Yaskawa INFORM job: CONTOUR2.JBI

/JOB
//NAME CONTOUR2
//POS
///NPOS 9848,0,0,0,0,0
///TOOL 0
///POSTYPE PULSE
///PULSE
C00000=-41004,59868,4099,4900,-34257,16705
C00001=-41004,59868,1099,4900,-34257,16705
C00002=-41004,64596,1380,5213,-31659,16463
C00003=-41004,59868,1099,4900,-34257,16705
C00004=-41004,59868,9099,4900,-34257,16705
C00005=3811,31631,-25134,676,-27450,-2228
C00006=3865,31716,-25032,668,-27483,-2249
C00007=3865,31716,-29032,668,-27483,-2249
C00008=3835,31810,-28918,671,-27518,-2237
C00009=3597,31820,-28908,705,-27519,-2144
C00010=3355,31766,-28975,741,-27496,-2051
C00011=3123,31694,-29064,775,-27467,-1961
C00012=2902,31602,-29176,808,-27431,-1876
C00013=2696,31482,-29322,839,-27385,-1796
C00014=2515,31319,-29520,866,-27323,-1727
C00015=2374,31161,-29713,888,-27263,-1673
C00016=2389,31321,-29519,885,-27322,-1678
C00017=2255,31496,-29308,902,-27386,-1624
C00018=2187,31630,-29147,910,-27435,-1597
C00019=2310,31450,-29364,894,-27369,-1646
C00020=2453,31290,-29556,876,-27311,-1703
C00021=2629,31465,-29344,848,-27378,-1770
C00022=2553,31625,-29151,858,-27436,-1740
C00023=2441,31812,-28926,872,-27504,-1694
C00024=2353,32012,-28684,882,-27578,-1659
C00025=2314,32240,-28409,885,-27661,-1642
C00026=2304,32475,-28124,884,-27749,-1636
C00027=2314,32706,-27845,880,-27834,-1639
C00028=2326,32679,-27878,879,-27824,-1644
C00029=2316,32448,-28157,883,-27739,-1641
C00030=2336,32210,-28445,883,-27651,-1651
C00031=2378,31984,-28718,879,-27567,-1669
C00032=2473,31787,-28955,867,-27496,-1707
C00033=2590,31603,-29177,853,-27428,-1754
C00034=2757,31554,-29235,829,-27412,-1819
C00035=2747,31685,-29077,829,-27460,-1815
C00036=2622,31865,-28860,845,-27526,-1765
C00037=2549,32074,-28608,854,-27603,-1735
C00038=2549,31957,-28749,855,-27559,-1736
C00039=2637,31757,-28991,844,-27486,-1771
C00040=2729,31601,-29178,833,-27429,-1808
C00041=2605,31782,-28960,849,-27495,-1759
C00042=2520,31985,-28716,859,-27569,-1724
C00043=2477,32210,-28444,863,-27652,-1706
C00044=2487,32441,-28165,859,-27738,-1708
C00045=2486,32674,-27883,856,-27824,-1706
C00046=2496,32905,-27604,853,-27910,-1708
C00047=2495,33138,-27322,850,-27996,-1706
C00048=2455,33357,-27057,854,-28077,-1689
C00049=2239,33295,-27134,885,-28051,-1605
C00050=2171,33103,-27367,896,-27979,-1580
C00051=2146,32876,-27642,902,-27895,-1572
C00052=2089,32656,-27907,913,-27813,-1551
C00053=2047,32433,-28178,921,-27730,-1537
C00054=2015,32207,-28451,928,-27646,-1526
C00055=2004,31976,-28730,933,-27561,-1523
C00056=2032,31743,-29011,931,-27475,-1536
C00057=2100,31532,-29266,924,-27397,-1564
C00058=2192,31334,-29505,913,-27325,-1601
C00059=2314,31152,-29724,897,-27259,-1650
C00060=2441,30973,-29940,881,-27194,-1701
C00061=2538,31160,-29713,865,-27264,-1737
C00062=2713,31335,-29500,838,-27330,-1804
C00063=2925,31445,-29366,806,-27373,-1885
C00064=3143,31543,-29246,774,-27412,-1970
C00065=3375,31616,-29157,739,-27441,-2059
C00066=3618,31670,-29089,704,-27463,-2153
C00067=3865,31716,-29032,668,-27483,-2249
C00068=3865,31716,-27632,668,-27483,-2249
C00069=3997,31675,-25080,649,-27469,-2301
C00070=3997,31675,-29080,649,-27469,-2301
C00071=3629,31643,-29122,703,-27453,-2158
C00072=3265,31552,-29234,756,-27416,-2017
C00073=3117,31368,-29458,779,-27346,-1961
C00074=2827,31365,-29463,821,-27343,-1848
C00075=2560,31123,-29757,862,-27250,-1746
C00076=2498,30791,-30159,875,-27127,-1724
C00077=2587,30462,-30556,865,-27006,-1761
C00078=2678,30133,-30954,855,-26885,-1799
C00079=2799,29820,-31331,841,-26770,-1848
C00080=2795,29751,-31415,842,-26744,-1847
C00081=2700,29995,-31120,854,-26834,-1808
C00082=2657,29651,-31536,864,-26706,-1794
C00083=2597,29318,-31939,876,-26583,-1774
C00084=2683,28990,-32335,867,-26462,-1809
C00085=2723,28642,-32756,865,-26333,-1827
C00086=2815,28557,-32857,852,-26303,-1863
C00087=2847,28244,-33236,851,-26187,-1878
C00088=2952,27925,-33622,839,-26069,-1921
C00089=3213,27690,-33905,802,-25984,-2023
C00090=3033,27904,-33647,827,-26062,-1952
C00091=2962,28220,-33265,834,-26179,-1922
C00092=2963,28089,-33423,835,-26130,-1924
C00093=3143,27897,-33654,810,-26061,-1995
C00094=3098,28244,-33236,814,-26189,-1975
C00095=3076,28338,-33122,816,-26223,-1966
C00096=3042,28684,-32704,817,-26351,-1950
C00097=3058,29035,-32280,811,-26481,-1954
C00098=3108,29326,-31927,801,-26589,-1971
C00099=3276,29624,-31566,773,-26701,-2034
C00100=3295,29634,-31554,770,-26705,-2041
C00101=3459,29782,-31375,745,-26761,-2103
C00102=3564,30094,-30996,726,-26878,-2142
C00103=3359,30318,-30727,754,-26959,-2061
C00104=3037,30467,-30548,800,-27011,-1935
C00105=3111,30271,-30785,791,-26939,-1965
C00106=3111,29941,-31184,794,-26817,-1968
C00107=3089,29614,-31579,801,-26696,-1962
C00108=3061,29461,-31764,806,-26639,-1952
C00109=3123,29801,-31353,794,-26765,-1974
C00110=3092,30139,-30945,795,-26890,-1959
C00111=2965,30424,-30600,810,-26995,-1908
C00112=2876,30690,-30279,821,-27093,-1872
C00113=2659,30936,-29983,850,-27182,-1786
C00114=2871,30740,-30218,821,-27111,-1869
C00115=3081,30482,-30530,793,-27018,-1953
C00116=3405,30337,-30703,747,-26967,-2079
C00117=3629,30413,-30610,714,-26997,-2165
C00118=3603,30113,-30974,720,-26885,-2157
C00119=3702,29893,-31239,708,-26804,-2197
C00120=4073,29908,-31220,653,-26812,-2340
C00121=4409,29785,-31366,605,-26769,-2471
C00122=4667,29549,-31651,569,-26683,-2572
C00123=4682,29665,-31511,566,-26727,-2577
C00124=4727,30001,-31105,556,-26852,-2593
C00125=4672,30326,-30711,562,-26973,-2570
C00126=4650,30631,-30342,563,-27086,-2559
C00127=4609,30958,-29945,566,-27208,-2542
C00128=4531,31274,-29563,575,-27324,-2510
C00129=4306,31488,-29305,606,-27402,-2422
C00130=3997,31675,-29080,649,-27469,-2301
C00131=3997,31675,-27680,649,-27469,-2301
C00132=4043,31695,-25057,642,-27476,-2318
C00133=4043,31695,-29057,642,-27476,-2318
C00134=5780,31150,-29707,394,-27289,-2995
C00135=5625,31340,-29477,415,-27359,-2934
C00136=3945,31835,-28888,655,-27528,-2280
C00137=5709,31371,-29439,403,-27371,-2966
C00138=6652,32744,-27767,260,-27893,-3328
C00139=6753,34511,-25621,239,-28558,-3363
C00140=6453,36318,-23427,276,-29233,-3243
C00141=6578,35948,-23875,259,-29096,-3292
C00142=6792,34132,-26080,234,-28416,-3379
C00143=6645,32383,-28206,262,-27758,-3326
C00144=7120,32806,-27689,192,-27921,-3510
C00145=6925,34048,-26182,216,-28386,-3431
C00146=6644,35901,-23931,250,-29079,-3318
C00147=5803,37019,-22583,363,-29488,-2986
C00148=3963,36746,-22938,616,-29357,-2262
C00149=2129,36463,-23304,868,-29224,-1540
C00150=289,36189,-23660,1121,-29094,-816
C00151=213,34463,-25744,1154,-28457,-802
C00152=323,33186,-27283,1156,-27988,-857
C00153=1338,31882,-28849,1029,-27519,-1265
C00154=2465,30575,-30421,882,-27047,-1713
C00155=1969,32162,-28506,936,-27629,-1508
C00156=1600,32867,-27657,980,-27886,-1359
C00157=996,33032,-27463,1063,-27939,-1121
C00158=1818,33311,-27119,944,-28052,-1440
C00159=1626,33396,-27018,970,-28081,-1365
C00160=1314,33620,-26749,1011,-28160,-1241
C00161=796,33812,-26524,1082,-28224,-1036
C00162=1636,32812,-27724,976,-27865,-1373
C00163=721,33056,-27436,1102,-27945,-1014
C00164=1464,34245,-25993,983,-28393,-1295
C00165=1936,35230,-24798,907,-28764,-1473
C00166=2213,35790,-24117,863,-28976,-1578
C00167=3722,35571,-24365,657,-28916,-2172
C00168=4244,35600,-24324,585,-28934,-2377
C00169=2395,35403,-24583,842,-28835,-1652
C00170=3210,35322,-24671,730,-28816,-1972
C00171=3567,35347,-24638,680,-28830,-2113
C00172=2031,34952,-25133,897,-28662,-1512
C00173=3721,35166,-23455,660,-28765,-2174
C00174=-41004,59868,4099,4900,-34257,16705
C00175=-41004,59868,1099,4900,-34257,16705
C00176=-41004,64596,1380,5213,-31659,16463
C00177=-41004,59868,1099,4900,-34257,16705
C00178=-41004,59868,9099,4900,-34257,16705
C00179=3721,35166,-20855,660,-28765,-2174
C00180=3721,35166,-24855,660,-28765,-2174
C00181=2130,35067,-24992,882,-28706,-1550
C00182=3955,35232,-24773,627,-28793,-2265
C00183=5703,35515,-24411,383,-28922,-2950
C00184=5623,36481,-23238,390,-29283,-2916
C00185=6165,34818,-25253,321,-28666,-3133
C00186=6218,33011,-27446,321,-27989,-3159
C00187=5066,32366,-28237,490,-27736,-2713
C00188=6014,32285,-28329,354,-27715,-3082
C00189=4649,33272,-27142,543,-28070,-2546
C00190=3598,34047,-26212,686,-28347,-2132
C00191=3164,33192,-27250,755,-28024,-1967
C00192=4473,31982,-28706,578,-27588,-2484
C00193=6195,31948,-28737,329,-27591,-3153
C00194=6280,32014,-28656,317,-27616,-3186
C00195=4570,31861,-28851,565,-27544,-2522
C00196=4080,32067,-28606,634,-27615,-2331
C00197=3506,32938,-27555,709,-27934,-2102
C00198=3001,33034,-27443,780,-27963,-1905
C00199=2855,33000,-27485,801,-27949,-1848
C00200=4043,31695,-29057,642,-27476,-2318
C00201=4043,31695,-27657,642,-27476,-2318
C00202=4163,31799,-24930,624,-27516,-2364
C00203=4163,31799,-28930,624,-27516,-2364
C00204=4084,31834,-28888,635,-27529,-2334
C00205=4008,31876,-28837,646,-27544,-2304
C00206=3930,31915,-28790,657,-27557,-2273
C00207=3853,31954,-28744,668,-27571,-2243
C00208=3786,32011,-28676,677,-27591,-2217
C00209=3763,32036,-28645,680,-27601,-2208
C00210=3832,31988,-28702,670,-27584,-2235
C00211=3909,31948,-28751,659,-27569,-2265
C00212=3987,31909,-28797,649,-27556,-2295
C00213=4064,31869,-28845,638,-27542,-2325
C00214=4142,31831,-28890,627,-27528,-2356
C00215=4222,31800,-28928,616,-27517,-2387
C00216=4302,31768,-28966,604,-27506,-2419
C00217=4382,31737,-29004,593,-27495,-2450
C00218=4465,31712,-29033,581,-27487,-2482
C00219=4547,31688,-29062,569,-27479,-2514
C00220=4630,31664,-29090,558,-27471,-2547
C00221=4713,31639,-29120,546,-27462,-2579
C00222=4798,31621,-29141,534,-27456,-2612
C00223=4883,31604,-29161,522,-27450,-2645
C00224=4968,31586,-29182,509,-27445,-2678
C00225=5053,31569,-29203,497,-27439,-2711
C00226=5140,31557,-29217,485,-27435,-2745
C00227=5225,31540,-29237,472,-27430,-2778
C00228=5314,31534,-29244,459,-27428,-2813
C00229=5403,31528,-29251,447,-27427,-2847
C00230=5495,31531,-29246,433,-27429,-2883
C00231=5589,31545,-29228,419,-27435,-2919
C00232=5684,31559,-29211,406,-27441,-2956
C00233=5773,31582,-29183,392,-27450,-2991
C00234=5862,31604,-29155,379,-27459,-3025
C00235=5946,31635,-29117,367,-27472,-3058
C00236=6027,31672,-29072,355,-27486,-3089
C00237=6103,31716,-29019,344,-27503,-3118
C00238=6174,31767,-28957,333,-27523,-3145
C00239=6196,31760,-28964,330,-27521,-3154
C00240=6126,31707,-29029,341,-27500,-3127
C00241=6052,31660,-29086,352,-27482,-3098
C00242=5973,31620,-29135,363,-27466,-3068
C00243=5890,31589,-29174,376,-27454,-3036
C00244=5800,31566,-29202,389,-27445,-3001
C00245=5711,31544,-29229,402,-27435,-2967
C00246=5616,31530,-29247,416,-27430,-2930
C00247=5522,31516,-29264,429,-27424,-2893
C00248=5427,31502,-29281,443,-27418,-2857
C00249=5338,31509,-29274,456,-27419,-2822
C00250=5249,31515,-29267,469,-27421,-2788
C00251=5162,31526,-29254,482,-27424,-2754
C00252=5077,31544,-29233,494,-27430,-2721
C00253=4992,31561,-29213,506,-27435,-2687
C00254=4907,31578,-29192,518,-27441,-2654
C00255=4822,31596,-29172,530,-27447,-2621
C00256=4736,31613,-29152,543,-27452,-2588
C00257=4652,31631,-29130,555,-27458,-2555
C00258=4569,31655,-29101,567,-27467,-2523
C00259=4486,31680,-29072,578,-27475,-2491
C00260=4404,31704,-29043,590,-27483,-2458
C00261=4323,31734,-29007,602,-27494,-2427
C00262=4241,31761,-28975,613,-27503,-2395
C00263=4163,31799,-28930,624,-27516,-2364
C00264=4163,31799,-27530,624,-27516,-2364
C00265=4231,31880,-24831,614,-27547,-2390
C00266=4231,31880,-28831,614,-27547,-2390
C00267=4158,31906,-28799,624,-27556,-2362
C00268=4087,31940,-28759,634,-27568,-2334
C00269=4017,31974,-28719,644,-27580,-2307
C00270=3946,32007,-28678,654,-27592,-2279
C00271=3878,32048,-28629,663,-27606,-2252
C00272=3808,32082,-28589,673,-27618,-2225
C00273=3738,32118,-28546,683,-27631,-2197
C00274=3669,32157,-28500,692,-27645,-2170
C00275=3604,32205,-28442,701,-27662,-2145
C00276=3536,32245,-28393,711,-27676,-2118
C00277=3474,32295,-28333,719,-27694,-2094
C00278=3419,32349,-28269,726,-27713,-2072
C00279=3360,32401,-28207,734,-27732,-2048
C00280=3308,32456,-28140,741,-27752,-2028
C00281=3261,32514,-28070,747,-27773,-2009
C00282=3215,32573,-27999,753,-27795,-1991
C00283=3179,32637,-27922,758,-27818,-1976
C00284=3142,32701,-27845,763,-27841,-1962
C00285=3098,32760,-27773,768,-27863,-1944
C00286=3061,32824,-27696,773,-27886,-1929
C00287=3041,32881,-27628,775,-27907,-1921
C00288=3081,32819,-27702,770,-27885,-1937
C00289=3124,32759,-27775,765,-27863,-1954
C00290=3163,32696,-27850,760,-27840,-1970
C00291=3200,32632,-27927,755,-27816,-1985
C00292=3245,32573,-27999,749,-27795,-2002
C00293=3289,32514,-28070,743,-27773,-2020
C00294=3341,32458,-28137,737,-27753,-2041
C00295=3393,32403,-28204,730,-27733,-2061
C00296=3451,32351,-28266,722,-27715,-2084
C00297=3510,32299,-28328,714,-27696,-2108
C00298=3576,32251,-28386,705,-27679,-2133
C00299=3643,32209,-28436,695,-27664,-2160
C00300=3709,32162,-28492,686,-27647,-2186
C00301=3777,32122,-28541,677,-27633,-2213
C00302=3847,32088,-28582,667,-27621,-2240
C00303=3916,32047,-28631,658,-27606,-2267
C00304=3986,32013,-28671,648,-27595,-2294
C00305=4054,31973,-28720,638,-27580,-2321
C00306=4125,31939,-28760,628,-27568,-2349
C00307=4198,31912,-28792,618,-27559,-2377
C00308=4269,31880,-28831,608,-27548,-2405
C00309=4342,31852,-28864,598,-27538,-2434
C00310=4415,31824,-28897,588,-27528,-2462
C00311=4486,31792,-28936,578,-27517,-2490
C00312=4559,31765,-28968,567,-27508,-2519
C00313=4633,31739,-29000,557,-27498,-2547
C00314=4707,31714,-29029,546,-27490,-2576
C00315=4782,31693,-29054,535,-27483,-2605
C00316=4856,31668,-29083,525,-27474,-2634
C00317=4895,31655,-29099,519,-27470,-2650
C00318=4818,31667,-29085,531,-27474,-2619
C00319=4743,31690,-29058,541,-27481,-2590
C00320=4668,31713,-29030,552,-27489,-2561
C00321=4594,31736,-29004,562,-27497,-2532
C00322=4521,31763,-28971,573,-27507,-2504
C00323=4448,31791,-28937,583,-27516,-2475
C00324=4375,31820,-28903,593,-27526,-2447
C00325=4302,31846,-28871,604,-27535,-2418
C00326=4231,31880,-28831,614,-27547,-2390
C00327=4231,31880,-27431,614,-27547,-2390
C00328=3770,31874,-24841,680,-27541,-2211
C00329=3770,31874,-28841,680,-27541,-2211
C00330=3645,31974,-28721,697,-27577,-2162
C00331=3526,32078,-28596,713,-27614,-2115
C00332=3408,32182,-28471,729,-27651,-2069
C00333=3304,32293,-28337,743,-27692,-2027
C00334=3202,32405,-28202,757,-27732,-1987
C00335=3117,32527,-28055,768,-27777,-1953
C00336=3034,32650,-27907,779,-27821,-1920
C00337=2951,32773,-27759,789,-27866,-1887
C00338=2874,32899,-27607,799,-27912,-1856
C00339=2812,33033,-27445,806,-27961,-1831
C00340=2711,33144,-27312,820,-28001,-1791
C00341=2574,33214,-27229,838,-28025,-1737
C00342=2507,33227,-27214,848,-28029,-1710
C00343=2511,33068,-27406,849,-27971,-1713
C00344=2515,32910,-27597,850,-27912,-1716
C00345=2519,32751,-27789,851,-27853,-1718
C00346=2513,32595,-27978,853,-27795,-1717
C00347=2507,32439,-28167,856,-27737,-1716
C00348=2501,32283,-28356,858,-27679,-1715
C00349=2534,32133,-27137,855,-27624,-1729
C00350=-41004,59868,4099,4900,-34257,16705
C00351=-41004,59868,1099,4900,-34257,16705
C00352=-41004,64596,1380,5213,-31659,16463
C00353=-41004,59868,1099,4900,-34257,16705
C00354=-41004,59868,9099,4900,-34257,16705
C00355=2534,32133,-24537,855,-27624,-1729
C00356=2534,32133,-28537,855,-27624,-1729
C00357=2586,31993,-28705,849,-27573,-1750
C00358=2645,31857,-28870,842,-27523,-1774
C00359=2728,31734,-29018,831,-27478,-1807
C00360=2832,31623,-29152,818,-27438,-1848
C00361=2866,31690,-29069,812,-27464,-1861
C00362=2793,31819,-28915,821,-27510,-1831
C00363=2730,31953,-28753,829,-27560,-1806
C00364=2678,32093,-28584,835,-27611,-1785
C00365=2654,32249,-28396,837,-27668,-1774
C00366=2656,32406,-28206,835,-27727,-1774
C00367=2666,32561,-28018,832,-27784,-1777
C00368=2672,32717,-27829,829,-27842,-1778
C00369=2668,32875,-27638,829,-27901,-1775
C00370=2690,32929,-27573,825,-27921,-1784
C00371=2687,32772,-27763,827,-27863,-1784
C00372=2681,32616,-27951,829,-27805,-1782
C00373=2675,32460,-28140,832,-27747,-1781
C00374=2669,32304,-28329,834,-27689,-1780
C00375=2684,32143,-28524,834,-27629,-1787
C00376=2728,31998,-28698,829,-27576,-1805
C00377=2790,31864,-28860,821,-27527,-1830
C00378=2862,31735,-29016,812,-27480,-1859
C00379=2968,31652,-29115,798,-27450,-1901
C00380=3115,31719,-29033,776,-27477,-1957
C00381=3130,31808,-28925,773,-27510,-1963
C00382=3056,31937,-28770,782,-27557,-1933
C00383=3003,32077,-28601,788,-27608,-1912
C00384=3023,32069,-28611,786,-27605,-1919
C00385=3076,31929,-28779,779,-27554,-1941
C00386=3151,31801,-28933,770,-27508,-1971
C00387=3281,31784,-28954,751,-27502,-2022
C00388=3392,31835,-28890,735,-27523,-2064
C00389=3297,31952,-28750,748,-27565,-2027
C00390=3244,32092,-28581,754,-27616,-2005
C00391=3254,32180,-28475,752,-27649,-2009
C00392=3279,32024,-28663,749,-27592,-2019
C00393=3353,31896,-28818,740,-27544,-2049
C00394=3471,31821,-28907,724,-27518,-2095
C00395=3642,31846,-28876,699,-27529,-2162
C00396=3770,31874,-28841,680,-27541,-2211
C00397=3770,31874,-27441,680,-27541,-2211
C00398=3508,31855,-24865,718,-27531,-2110
C00399=3508,31855,-28865,718,-27531,-2110
C00400=3499,31854,-28868,719,-27530,-2106
C00401=3489,31852,-28869,721,-27530,-2102
C00402=3481,31858,-28862,722,-27532,-2099
C00403=3471,31859,-28861,723,-27532,-2095
C00404=3463,31863,-28857,724,-27533,-2092
C00405=3455,31868,-28850,726,-27535,-2089
C00406=3447,31874,-28843,727,-27537,-2085
C00407=3439,31880,-28836,728,-27540,-2082
C00408=3431,31886,-28829,729,-27542,-2079
C00409=3423,31892,-28822,730,-27544,-2076
C00410=3415,31897,-28815,731,-27546,-2073
C00411=3413,31906,-28804,731,-27549,-2072
C00412=3406,31913,-28797,732,-27551,-2069
C00413=3398,31919,-28790,733,-27554,-2066
C00414=3390,31925,-28782,734,-27556,-2063
C00415=3389,31934,-28771,734,-27559,-2062
C00416=3381,31940,-28764,736,-27561,-2059
C00417=3378,31949,-28753,736,-27564,-2058
C00418=3371,31955,-28745,737,-27567,-2056
C00419=3366,31963,-28736,737,-27570,-2054
C00420=3365,31973,-28725,737,-27573,-2053
C00421=3364,31982,-28713,738,-27577,-2053
C00422=3360,31990,-28704,738,-27580,-2051
C00423=3353,31996,-28696,739,-27582,-2048
C00424=3352,32006,-28684,739,-27586,-2048
C00425=3351,32016,-28672,739,-27589,-2047
C00426=3350,32026,-28660,739,-27593,-2047
C00427=3349,32035,-28649,739,-27596,-2046
C00428=3348,32045,-28637,739,-27600,-2046
C00429=3347,32055,-28625,739,-27604,-2046
C00430=3349,32059,-28620,739,-27605,-2047
C00431=3357,32053,-28627,738,-27603,-2050
C00432=3358,32043,-28639,738,-27599,-2050
C00433=3359,32034,-28651,738,-27596,-2051
C00434=3360,32024,-28663,738,-27592,-2051
C00435=3362,32015,-28674,738,-27589,-2052
C00436=3370,32009,-28681,736,-27587,-2055
C00437=3373,32000,-28691,736,-27583,-2056
C00438=3374,31990,-28703,736,-27580,-2056
C00439=3375,31980,-28715,736,-27576,-2057
C00440=3376,31971,-28727,736,-27573,-2057
C00441=3383,31964,-28734,735,-27570,-2060
C00442=3387,31957,-28744,734,-27568,-2062
C00443=3392,31949,-28753,734,-27565,-2064
C00444=3399,31943,-28761,733,-27562,-2066
C00445=3401,31934,-28772,733,-27559,-2067
C00446=3409,31928,-28779,732,-27557,-2071
C00447=3417,31922,-28785,730,-27555,-2074
C00448=3422,31914,-28795,730,-27552,-2076
C00449=3426,31907,-28804,729,-27549,-2077
C00450=3434,31901,-28811,728,-27547,-2080
C00451=3442,31895,-28818,727,-27545,-2084
C00452=3450,31889,-28825,726,-27543,-2087
C00453=3458,31883,-28832,725,-27541,-2090
C00454=3466,31877,-28839,724,-27539,-2093
C00455=3474,31872,-28846,723,-27537,-2096
C00456=3482,31866,-28853,722,-27535,-2099
C00457=3491,31862,-28858,720,-27533,-2103
C00458=3500,31861,-28858,719,-27533,-2106
C00459=3508,31855,-28865,718,-27531,-2110
C00460=3508,31855,-27465,718,-27531,-2110
C00461=3267,31838,-24888,753,-27522,-2016
C00462=3267,31838,-28888,753,-27522,-2016
C00463=3270,31811,-28921,753,-27512,-2017
C00464=3247,31841,-28885,756,-27523,-2008
C00465=3224,31871,-28848,759,-27534,-1999
C00466=3204,31903,-28810,761,-27546,-1991
C00467=3187,31937,-28769,763,-27558,-1984
C00468=3171,31971,-28728,765,-27571,-1978
C00469=3151,32003,-28689,768,-27582,-1970
C00470=3138,32039,-28646,769,-27596,-1964
C00471=3133,32079,-28598,770,-27610,-1962
C00472=3119,32114,-28555,771,-27623,-1957
C00473=3106,32150,-28512,773,-27636,-1951
C00474=3086,32182,-28473,776,-27648,-1943
C00475=3069,32216,-28432,778,-27660,-1936
C00476=3054,32250,-28391,780,-27673,-1930
C00477=3033,32282,-28353,782,-27684,-1922
C00478=3010,32312,-28317,785,-27695,-1913
C00479=2995,32346,-28275,787,-27708,-1906
C00480=2973,32377,-28238,790,-27719,-1898
C00481=2960,32413,-28195,791,-27733,-1893
C00482=2937,32443,-28158,794,-27743,-1883
C00483=2916,32475,-28121,797,-27755,-1875
C00484=2897,32507,-28082,800,-27767,-1867
C00485=2877,32539,-28043,802,-27778,-1859
C00486=2855,32569,-28006,805,-27789,-1851
C00487=2838,32603,-27966,807,-27802,-1844
C00488=2819,32635,-27927,809,-27813,-1836
C00489=2806,32671,-27884,811,-27826,-1831
C00490=2786,32703,-27845,813,-27838,-1823
C00491=2770,32737,-27805,815,-27850,-1816
C00492=2757,32772,-27762,817,-27864,-1811
C00493=2759,32802,-27725,816,-27875,-1812
C00494=2777,32770,-27765,814,-27863,-1819
C00495=2791,32734,-27807,812,-27850,-1825
C00496=2810,32702,-27846,810,-27838,-1832
C00497=2826,32668,-27887,808,-27826,-1839
C00498=2843,32634,-27928,806,-27813,-1845
C00499=2862,32602,-27966,804,-27802,-1853
C00500=2882,32570,-28005,801,-27790,-1861
C00501=2898,32537,-28046,799,-27778,-1868
C00502=2921,32506,-28082,796,-27767,-1877
C00503=2940,32474,-28121,794,-27755,-1885
C00504=2960,32442,-28160,791,-27743,-1892
C00505=2980,32410,-28198,788,-27732,-1901
C00506=2994,32375,-28241,787,-27719,-1906
C00507=3017,32345,-28277,784,-27708,-1915
C00508=3039,32314,-28314,781,-27697,-1924
C00509=3053,32279,-28356,779,-27684,-1930
C00510=3076,32249,-28393,776,-27673,-1939
C00511=3091,32214,-28435,775,-27660,-1945
C00512=3111,32182,-28473,772,-27648,-1953
C00513=3117,32142,-28521,772,-27634,-1955
C00514=3137,32110,-28560,769,-27622,-1963
C00515=3144,32071,-28607,768,-27608,-1966
C00516=3157,32035,-28650,767,-27594,-1972
C00517=3171,32000,-28693,765,-27581,-1977
C00518=3189,31967,-28733,763,-27569,-1984
C00519=3207,31934,-28772,761,-27557,-1992
C00520=3221,31899,-28815,759,-27544,-1998
C00521=3244,31868,-28851,756,-27533,-2007
C00522=3267,31838,-27488,753,-27522,-2016
C00523=-41004,59868,4099,4900,-34257,16705
C00524=-41004,59868,1099,4900,-34257,16705
C00525=-41004,64596,1380,5213,-31659,16463
C00526=-41004,59868,1099,4900,-34257,16705
C00527=-41004,59868,9099,4900,-34257,16705
C00528=3267,31838,-24888,753,-27522,-2016
C00529=3267,31838,-28888,753,-27522,-2016
C00530=3267,31838,-27488,753,-27522,-2016
C00531=2965,31780,-24961,797,-27498,-1899
C00532=2965,31780,-28961,797,-27498,-1899
C00533=2972,31757,-28988,796,-27489,-1902
C00534=2986,31738,-29011,794,-27482,-1907
C00535=3000,31719,-29034,792,-27475,-1913
C00536=2997,31704,-29052,793,-27470,-1912
C00537=2985,31724,-29028,795,-27477,-1907
C00538=2969,31742,-29006,797,-27484,-1900
C00539=2961,31764,-28979,798,-27492,-1897
C00540=2947,31784,-28956,799,-27499,-1892
C00541=2937,31805,-28931,801,-27507,-1887
C00542=2925,31825,-28906,802,-27514,-1883
C00543=2919,31849,-28878,803,-27523,-1880
C00544=2910,31871,-28851,804,-27531,-1877
C00545=2898,31891,-28827,805,-27538,-1872
C00546=2886,31911,-28803,807,-27546,-1867
C00547=2884,31936,-28772,807,-27555,-1866
C00548=2872,31957,-28747,808,-27562,-1861
C00549=2860,31977,-28723,810,-27570,-1857
C00550=2855,32001,-28694,810,-27579,-1855
C00551=2846,32022,-28668,812,-27586,-1851
C00552=2841,32047,-28639,812,-27595,-1849
C00553=2831,32068,-28613,813,-27603,-1845
C00554=2827,32092,-28583,814,-27612,-1843
C00555=2817,32114,-28558,815,-27620,-1839
C00556=2815,32139,-28527,815,-27630,-1838
C00557=2803,32160,-28502,816,-27637,-1833
C00558=2800,32185,-28472,816,-27646,-1832
C00559=2789,32205,-28447,818,-27654,-1827
C00560=2786,32231,-28416,818,-27663,-1826
C00561=2774,32251,-28392,820,-27670,-1821
C00562=2772,32276,-28361,820,-27680,-1820
C00563=2770,32302,-28330,820,-27689,-1819
C00564=2758,32322,-28306,821,-27697,-1814
C00565=2755,32348,-28275,821,-27706,-1813
C00566=2759,32363,-28257,821,-27712,-1815
C00567=2766,32340,-28285,820,-27703,-1818
C00568=2778,32320,-28309,818,-27696,-1822
C00569=2780,32294,-28340,818,-27686,-1823
C00570=2792,32274,-28364,817,-27679,-1828
C00571=2795,32248,-28395,817,-27670,-1829
C00572=2807,32228,-28419,815,-27662,-1834
C00573=2809,32203,-28450,815,-27653,-1835
C00574=2821,32182,-28475,814,-27646,-1840
C00575=2823,32157,-28505,813,-27636,-1841
C00576=2830,32134,-28533,813,-27628,-1844
C00577=2837,32111,-28561,812,-27619,-1847
C00578=2844,32088,-28588,811,-27611,-1850
C00579=2852,32066,-28616,810,-27603,-1853
C00580=2859,32043,-28643,810,-27594,-1856
C00581=2866,32020,-28671,809,-27586,-1859
C00582=2873,31997,-28699,808,-27577,-1861
C00583=2880,31974,-28726,807,-27569,-1864
C00584=2892,31954,-28750,806,-27562,-1869
C00585=2901,31932,-28777,805,-27554,-1873
C00586=2908,31909,-28804,804,-27545,-1876
C00587=2919,31888,-28830,802,-27537,-1880
C00588=2930,31867,-28855,801,-27530,-1884
C00589=2933,31842,-28885,801,-27521,-1886
C00590=2945,31822,-28909,799,-27513,-1891
C00591=2957,31802,-28934,798,-27506,-1895
C00592=2965,31780,-28961,797,-27498,-1899
C00593=2965,31780,-27561,797,-27498,-1899
C00594=2344,31645,-25127,888,-27442,-1658
C00595=2344,31645,-29127,888,-27442,-1658
C00596=2356,31620,-29158,886,-27433,-1663
C00597=2368,31595,-29188,885,-27423,-1668
C00598=2384,31572,-29215,883,-27415,-1674
C00599=2402,31550,-29242,880,-27407,-1681
C00600=2414,31525,-29272,879,-27398,-1686
C00601=2431,31503,-29299,877,-27390,-1693
C00602=2449,31481,-29326,874,-27382,-1700
C00603=2467,31459,-29352,872,-27374,-1707
C00604=2484,31437,-29379,870,-27366,-1714
C00605=2484,31419,-29400,870,-27359,-1714
C00606=2467,31441,-29374,872,-27367,-1707
C00607=2449,31463,-29347,874,-27375,-1700
C00608=2428,31483,-29323,877,-27383,-1692
C00609=2413,31507,-29294,879,-27391,-1686
C00610=2394,31528,-29269,882,-27399,-1678
C00611=2378,31551,-29241,884,-27407,-1672
C00612=2360,31573,-29215,886,-27415,-1665
C00613=2342,31595,-29188,888,-27423,-1658
C00614=2331,31621,-29157,890,-27432,-1653
C00615=2313,31643,-29131,892,-27440,-1646
C00616=2303,31668,-29100,893,-27450,-1642
C00617=2289,31693,-29070,895,-27459,-1636
C00618=2281,31720,-29038,896,-27469,-1633
C00619=2274,31748,-29003,896,-27479,-1630
C00620=2262,31773,-28973,898,-27488,-1625
C00621=2250,31798,-28943,899,-27497,-1620
C00622=2244,31827,-28909,900,-27508,-1618
C00623=2235,31854,-28876,901,-27518,-1614
C00624=2223,31879,-28846,902,-27527,-1609
C00625=2221,31909,-28809,902,-27538,-1608
C00626=2208,31934,-28779,904,-27547,-1603
C00627=2206,31965,-28742,904,-27559,-1602
C00628=2203,31995,-28705,904,-27570,-1601
C00629=2201,32026,-28669,904,-27581,-1600
C00630=2198,32056,-28632,904,-27592,-1598
C00631=2196,32087,-28595,904,-27604,-1597
C00632=2193,32117,-28558,904,-27615,-1596
C00633=2191,32147,-28522,904,-27626,-1595
C00634=2188,32178,-28485,904,-27637,-1594
C00635=2202,32195,-28464,902,-27644,-1599
C00636=2209,32167,-28497,901,-27634,-1602
C00637=2212,32137,-28534,901,-27622,-1603
C00638=2214,32107,-28571,901,-27611,-1604
C00639=2217,32076,-28608,901,-27600,-1605
C00640=2216,32046,-28644,901,-27589,-1605
C00641=2212,32018,-28678,902,-27578,-1604
C00642=2217,31989,-28713,902,-27568,-1606
C00643=2226,31962,-28745,901,-27558,-1610
C00644=2232,31934,-28780,900,-27547,-1612
C00645=2241,31907,-28812,899,-27537,-1616
C00646=2247,31878,-28847,899,-27527,-1619
C00647=2256,31851,-28879,898,-27517,-1622
C00648=2268,31826,-28909,896,-27508,-1627
C00649=2273,31797,-28945,896,-27497,-1629
C00650=2283,31771,-28976,895,-27487,-1633
C00651=2295,31746,-29007,894,-27478,-1638
C00652=2305,31720,-29038,892,-27469,-1642
C00653=2316,31694,-29069,891,-27459,-1647
C00654=2327,31668,-29100,890,-27450,-1651
C00655=2344,31645,-29127,888,-27442,-1658
C00656=2344,31645,-27727,888,-27442,-1658
C00657=1836,31669,-25103,960,-27445,-1460
C00658=1836,31669,-29103,960,-27445,-1460
C00659=1828,31648,-29127,962,-27438,-1457
C00660=1816,31671,-29100,963,-27446,-1452
C00661=1810,31697,-29068,964,-27456,-1450
C00662=1802,31723,-29038,964,-27465,-1447
C00663=1800,31751,-29004,964,-27475,-1446
C00664=1798,31779,-28969,964,-27486,-1444
C00665=1796,31808,-28935,964,-27496,-1443
C00666=1793,31836,-28901,964,-27507,-1442
C00667=1791,31864,-28867,964,-27517,-1441
C00668=1789,31893,-28832,964,-27528,-1440
C00669=1787,31921,-28798,964,-27538,-1439
C00670=1786,31949,-28764,964,-27548,-1439
C00671=1793,31975,-28733,963,-27558,-1441
C00672=1791,32004,-28698,963,-27569,-1440
C00673=1799,32030,-28667,961,-27578,-1443
C00674=1806,32056,-28635,960,-27588,-1446
C00675=1811,32082,-28603,959,-27598,-1447
C00676=1816,32109,-28571,958,-27608,-1449
C00677=1821,32135,-28539,957,-27618,-1451
C00678=1829,32161,-28507,956,-27627,-1454
C00679=1839,32187,-28477,954,-27637,-1457
C00680=1845,32213,-28445,953,-27647,-1459
C00681=1853,32239,-28413,951,-27656,-1462
C00682=1861,32265,-28382,950,-27666,-1465
C00683=1873,32290,-28352,948,-27675,-1470
C00684=1885,32315,-28322,946,-27685,-1474
C00685=1890,32341,-28290,945,-27694,-1476
C00686=1902,32366,-28260,943,-27704,-1481
C00687=1911,32392,-28228,941,-27713,-1484
C00688=1919,32418,-28197,940,-27723,-1487
C00689=1932,32433,-28179,938,-27729,-1492
C00690=1929,32410,-28207,938,-27720,-1491
C00691=1921,32384,-28238,940,-27711,-1488
C00692=1913,32358,-28269,941,-27701,-1485
C00693=1905,32332,-28301,943,-27691,-1482
C00694=1897,32306,-28332,944,-27682,-1479
C00695=1890,32280,-28363,946,-27672,-1476
C00696=1879,32255,-28394,947,-27663,-1472
C00697=1874,32229,-28426,948,-27653,-1470
C00698=1866,32203,-27057,950,-27643,-1468
C00699=-41004,59868,4099,4900,-34257,16705
C00700=-41004,59868,1099,4900,-34257,16705
C00701=-41004,64596,1380,5213,-31659,16463
C00702=-41004,59868,1099,4900,-34257,16705
C00703=-41004,59868,9099,4900,-34257,16705
C00704=1866,32203,-24457,950,-27643,-1468
C00705=1866,32203,-28457,950,-27643,-1468
C00706=1856,32177,-28488,951,-27633,-1464
C00707=1850,32151,-28520,953,-27624,-1462
C00708=1842,32125,-28551,954,-27614,-1459
C00709=1833,32099,-28583,956,-27604,-1456
C00710=1825,32073,-28614,957,-27595,-1453
C00711=1824,32046,-28647,958,-27585,-1453
C00712=1819,32019,-28679,959,-27575,-1451
C00713=1812,31993,-28711,960,-27565,-1448
C00714=1809,31966,-28744,961,-27555,-1447
C00715=1806,31939,-28776,961,-27545,-1446
C00716=1808,31911,-28811,961,-27534,-1447
C00717=1801,31884,-28842,963,-27525,-1445
C00718=1802,31856,-28876,963,-27514,-1445
C00719=1804,31828,-28910,963,-27504,-1447
C00720=1806,31800,-28945,963,-27493,-1448
C00721=1808,31771,-28979,963,-27483,-1449
C00722=1811,31743,-29013,963,-27472,-1450
C00723=1822,31720,-29041,962,-27464,-1455
C00724=1825,31692,-29075,962,-27454,-1456
C00725=1836,31669,-29103,960,-27445,-1460
C00726=1836,31669,-27703,960,-27445,-1460
C00727=1675,31672,-25100,983,-27445,-1397
C00728=1675,31672,-29100,983,-27445,-1397
C00729=1677,31648,-29129,983,-27436,-1398
C00730=1678,31623,-29159,983,-27427,-1399
C00731=1680,31599,-29188,983,-27418,-1400
C00732=1682,31574,-29218,983,-27409,-1401
C00733=1684,31550,-29248,983,-27400,-1402
C00734=1686,31525,-29277,983,-27391,-1403
C00735=1688,31501,-29307,983,-27382,-1404
C00736=1696,31480,-29332,983,-27374,-1407
C00737=1701,31457,-29359,982,-27366,-1409
C00738=1703,31433,-29389,982,-27357,-1410
C00739=1713,31413,-29413,981,-27350,-1414
C00740=1719,31391,-29439,980,-27341,-1417
C00741=1737,31375,-29458,978,-27336,-1424
C00742=1749,31356,-29481,976,-27329,-1429
C00743=1757,31335,-29506,975,-27321,-1432
C00744=1770,31317,-29528,974,-27315,-1437
C00745=1784,31299,-29550,972,-27308,-1443
C00746=1796,31280,-29572,971,-27301,-1448
C00747=1809,31262,-29595,969,-27295,-1453
C00748=1821,31243,-29617,967,-27288,-1458
C00749=1840,31228,-29635,965,-27282,-1465
C00750=1851,31209,-29658,963,-27275,-1470
C00751=1863,31190,-29681,962,-27268,-1475
C00752=1875,31171,-29704,960,-27262,-1479
C00753=1886,31151,-29728,959,-27254,-1484
C00754=1898,31132,-29750,957,-27248,-1489
C00755=1910,31113,-29773,956,-27241,-1493
C00756=1917,31092,-29799,955,-27233,-1496
C00757=1923,31070,-29826,955,-27225,-1499
C00758=1910,31088,-29804,956,-27231,-1494
C00759=1897,31107,-29781,958,-27238,-1489
C00760=1885,31125,-29759,960,-27245,-1483
C00761=1872,31143,-29737,961,-27251,-1478
C00762=1859,31162,-29715,963,-27258,-1473
C00763=1846,31180,-29693,964,-27265,-1468
C00764=1833,31199,-29671,966,-27272,-1463
C00765=1820,31217,-29648,968,-27278,-1458
C00766=1808,31236,-29626,969,-27285,-1453
C00767=1788,31250,-29609,972,-27290,-1445
C00768=1776,31269,-29586,974,-27297,-1440
C00769=1762,31287,-29564,975,-27304,-1435
C00770=1750,31306,-29542,977,-27310,-1429
C00771=1741,31326,-29517,978,-27318,-1426
C00772=1730,31345,-29494,979,-27325,-1421
C00773=1718,31365,-29471,981,-27332,-1417
C00774=1705,31383,-29449,982,-27338,-1412
C00775=1695,31403,-29425,984,-27346,-1407
C00776=1683,31422,-29402,985,-27353,-1403
C00777=1681,31446,-29372,985,-27362,-1402
C00778=1680,31471,-29343,985,-27371,-1401
C00779=1678,31495,-29313,985,-27380,-1400
C00780=1676,31520,-29284,985,-27389,-1399
C00781=1674,31544,-29254,985,-27398,-1398
C00782=1672,31569,-29225,985,-27407,-1397
C00783=1671,31593,-29195,985,-27416,-1396
C00784=1669,31618,-29165,985,-27425,-1396
C00785=1667,31642,-29136,985,-27434,-1395
C00786=1665,31667,-29106,985,-27443,-1394
C00787=1663,31691,-29077,985,-27452,-1393
C00788=1675,31672,-29100,983,-27445,-1397
C00789=1675,31672,-27700,983,-27445,-1397
C00790=1603,31826,-24914,992,-27501,-1368
C00791=1603,31826,-28914,992,-27501,-1368
C00792=1593,31824,-28916,993,-27500,-1364
C00793=1592,31834,-28905,993,-27504,-1364
C00794=1592,31844,-28893,993,-27507,-1364
C00795=1591,31854,-28881,993,-27511,-1363
C00796=1590,31863,-28869,993,-27515,-1363
C00797=1589,31873,-28857,993,-27518,-1363
C00798=1590,31883,-28846,993,-27522,-1363
C00799=1597,31891,-28836,992,-27525,-1365
C00800=1598,31900,-28825,992,-27528,-1366
C00801=1597,31910,-28813,992,-27532,-1365
C00802=1596,31920,-28801,992,-27535,-1365
C00803=1602,31928,-28791,991,-27539,-1367
C00804=1605,31937,-28781,990,-27542,-1368
C00805=1604,31946,-28769,990,-27546,-1368
C00806=1608,31955,-28758,989,-27549,-1369
C00807=1613,31964,-28748,989,-27552,-1371
C00808=1614,31973,-28737,988,-27555,-1372
C00809=1621,31981,-28727,987,-27558,-1374
C00810=1621,31990,-28716,987,-27562,-1374
C00811=1620,32000,-28704,987,-27566,-1374
C00812=1620,32010,-28692,987,-27569,-1373
C00813=1626,32018,-28682,986,-27572,-1376
C00814=1628,32027,-28671,986,-27576,-1376
C00815=1633,32036,-28661,985,-27579,-1378
C00816=1637,32044,-28651,984,-27582,-1380
C00817=1636,32054,-28639,984,-27586,-1379
C00818=1639,32063,-28628,984,-27589,-1380
C00819=1645,32071,-28618,983,-27592,-1383
C00820=1645,32081,-28606,983,-27596,-1382
C00821=1651,32089,-28597,982,-27599,-1385
C00822=1659,32087,-28598,981,-27598,-1388
C00823=1662,32081,-28606,980,-27596,-1389
C00824=1655,32073,-28616,981,-27593,-1387
C00825=1656,32063,-28628,981,-27589,-1387
C00826=1656,32053,-28639,981,-27585,-1387
C00827=1650,32045,-28649,983,-27582,-1385
C00828=1648,32036,-28660,983,-27579,-1384
C00829=1648,32026,-28672,983,-27575,-1384
C00830=1644,32018,-28682,984,-27572,-1383
C00831=1640,32009,-28693,984,-27569,-1381
C00832=1640,32000,-28704,984,-27565,-1381
C00833=1638,31990,-28715,985,-27562,-1381
C00834=1632,31982,-28725,986,-27559,-1378
C00835=1632,31973,-28737,986,-27556,-1378
C00836=1625,31965,-28747,987,-27552,-1376
C00837=1624,31956,-28758,987,-27549,-1375
C00838=1624,31946,-28770,987,-27545,-1376
C00839=1619,31937,-28780,988,-27542,-1374
C00840=1616,31929,-28790,989,-27539,-1372
C00841=1616,31919,-28802,989,-27535,-1373
C00842=1613,31910,-28813,989,-27532,-1372
C00843=1607,31902,-28823,990,-27529,-1369
C00844=1608,31892,-28835,990,-27525,-1370
C00845=1609,31882,-28846,990,-27522,-1370
C00846=1610,31873,-28858,990,-27518,-1370
C00847=1609,31863,-28869,991,-27515,-1370
C00848=1602,31855,-28879,992,-27512,-1368
C00849=1602,31846,-28891,992,-27508,-1368
C00850=1602,31836,-28902,992,-27505,-1368
C00851=1603,31826,-28914,992,-27501,-1368
C00852=1603,31826,-27514,992,-27501,-1368
C00853=1374,31784,-24967,1025,-27483,-1279
C00854=1374,31784,-28967,1025,-27483,-1279
C00855=1299,31867,-28867,1035,-27513,-1249
C00856=1252,31966,-28748,1040,-27549,-1230
C00857=1191,32057,-28639,1048,-27582,-1206
C00858=1102,32133,-28548,1059,-27609,-1171
C00859=1015,32209,-28457,1071,-27636,-1136
C00860=910,32252,-28405,1085,-27651,-1095
C00861=801,32282,-28370,1100,-27661,-1052
C00862=702,32340,-28301,1114,-27681,-1013
C00863=613,32409,-28218,1126,-27705,-977
C00864=531,32488,-28124,1136,-27733,-944
C00865=466,32576,-28018,1144,-27765,-918
C00866=411,32670,-27905,1151,-27799,-896
C00867=366,32769,-27786,1156,-27835,-878
C00868=340,32879,-27654,1158,-27875,-866
C00869=305,32982,-27529,1161,-27913,-851
C00870=311,32870,-27665,1162,-27871,-855
C00871=318,32749,-27811,1163,-27827,-859
C00872=325,32628,-27956,1163,-27783,-863
C00873=331,32508,-28102,1164,-27738,-866
C00874=338,32387,-26847,1165,-27694,-870
C00875=-41004,59868,4099,4900,-34257,16705
C00876=-41004,59868,1099,4900,-34257,16705
C00877=-41004,64596,1380,5213,-31659,16463
C00878=-41004,59868,1099,4900,-34257,16705
C00879=-41004,59868,9099,4900,-34257,16705
C00880=338,32387,-24247,1165,-27694,-870
C00881=338,32387,-28247,1165,-27694,-870
C00882=345,32267,-28392,1165,-27650,-874
C00883=351,32146,-28538,1166,-27605,-878
C00884=358,32025,-28683,1167,-27561,-881
C00885=439,32000,-28714,1156,-27553,-913
C00886=565,32018,-28690,1137,-27561,-962
C00887=691,32037,-28667,1119,-27569,-1011
C00888=814,32045,-28656,1102,-27573,-1059
C00889=940,32063,-28633,1084,-27582,-1108
C00890=1063,32072,-28622,1066,-27586,-1156
C00891=1108,32059,-28636,1060,-27582,-1173
C00892=985,32051,-28647,1077,-27577,-1126
C00893=859,32032,-28671,1095,-27569,-1077
C00894=733,32014,-28694,1114,-27561,-1028
C00895=607,31996,-28717,1132,-27553,-979
C00896=484,31987,-28728,1149,-27549,-931
C00897=362,31961,-28761,1167,-27537,-884
C00898=368,31840,-28906,1168,-27493,-887
C00899=375,31720,-29052,1169,-27449,-891
C00900=382,31599,-29197,1169,-27405,-894
C00901=388,31479,-29343,1170,-27360,-898
C00902=395,31358,-29488,1171,-27316,-902
C00903=402,31237,-29634,1171,-27272,-906
C00904=408,31117,-29779,1172,-27227,-909
C00905=491,31192,-29688,1159,-27256,-941
C00906=560,31294,-29564,1148,-27294,-967
C00907=594,31405,-29430,1142,-27335,-979
C00908=617,31518,-29294,1137,-27377,-987
C00909=600,31633,-29155,1138,-27419,-979
C00910=533,31720,-29050,1146,-27451,-952
C00911=436,31785,-28973,1159,-27474,-914
C00912=468,31796,-28959,1154,-27478,-926
C00913=565,31731,-29037,1141,-27455,-965
C00914=620,31637,-29149,1135,-27421,-987
C00915=731,31632,-29155,1119,-27420,-1030
C00916=854,31659,-29121,1101,-27432,-1078
C00917=980,31678,-29097,1083,-27440,-1127
C00918=1103,31705,-29064,1065,-27451,-1174
C00919=1226,31713,-29053,1047,-27456,-1222
C00920=1349,31722,-29042,1029,-27460,-1270
C00921=1374,31784,-28967,1025,-27483,-1279
C00922=1374,31784,-27567,1025,-27483,-1279
C00923=1418,31602,-25186,1021,-27416,-1298
C00924=1418,31602,-29186,1021,-27416,-1298
C00925=980,31658,-29121,1083,-27433,-1127
C00926=632,31443,-29383,1136,-27350,-993
C00927=415,31001,-29919,1173,-27185,-913
C00928=442,30499,-30524,1176,-27000,-928
C00929=470,29997,-31129,1179,-26816,-944
C00930=833,30209,-30872,1123,-26897,-1083
C00931=1122,30591,-30409,1076,-27041,-1192
C00932=1333,30864,-30078,1042,-27143,-1271
C00933=842,30907,-30029,1113,-27154,-1080
C00934=534,31090,-29810,1154,-27219,-959
C00935=924,30924,-30008,1101,-27162,-1112
C00936=1399,30851,-30094,1033,-27139,-1297
C00937=1086,30540,-30471,1082,-27021,-1178
C00938=834,30136,-30960,1124,-26870,-1084
C00939=1197,29999,-31123,1073,-26823,-1226
C00940=1610,29915,-31222,1014,-26796,-1387
C00941=1773,30270,-30792,986,-26928,-1447
C00942=1905,30656,-30326,962,-27072,-1495
C00943=1799,30269,-30794,982,-26928,-1457
C00944=1996,30113,-30981,955,-26872,-1535
C00945=2168,30426,-30602,926,-26989,-1599
C00946=2168,30176,-30904,929,-26897,-1601
C00947=1771,29939,-31192,990,-26806,-1449
C00948=1298,29874,-31273,1060,-26778,-1266
C00949=945,30094,-31010,1108,-26856,-1127
C00950=542,29933,-31206,1169,-26793,-972
C00951=723,29701,-31485,1146,-26709,-1045
C00952=1220,29652,-31541,1074,-26695,-1238
C00953=1705,29652,-31539,1003,-26699,-1426
C00954=1719,29635,-31559,1001,-26693,-1431
C00955=1179,29548,-31667,1081,-26657,-1223
C00956=1092,29650,-31545,1093,-26693,-1188
C00957=593,29690,-31499,1165,-26704,-994
C00958=734,29495,-31734,1147,-26633,-1051
C00959=703,29479,-31753,1152,-26627,-1039
C00960=514,29209,-32080,1183,-26526,-968
C00961=542,28707,-32685,1186,-26342,-984
C00962=569,28205,-33290,1189,-26158,-999
C00963=597,27703,-33895,1192,-25973,-1015
C00964=909,27646,-33963,1147,-25954,-1136
C00965=1239,27952,-33594,1093,-26069,-1260
C00966=1696,27827,-33743,1027,-26026,-1437
C00967=1836,28233,-33253,1001,-26176,-1488
C00968=2058,28139,-33365,969,-26143,-1574
C00969=2120,28534,-32888,956,-26289,-1595
C00970=2454,28499,-32929,906,-26279,-1724
C00971=2660,28768,-32604,873,-26379,-1802
C00972=2558,29228,-32048,883,-26549,-1759
C00973=2625,29703,-31474,868,-26725,-1782
C00974=2633,30176,-30901,862,-26901,-1781
C00975=2401,30568,-30430,891,-27043,-1688
C00976=2004,30850,-30091,945,-27144,-1532
C00977=1639,31165,-29713,994,-27257,-1388
C00978=1236,31294,-29559,1051,-27301,-1230
C00979=1019,31027,-29883,1086,-27200,-1148
C00980=1519,31011,-29899,1014,-27199,-1342
C00981=1491,30997,-29916,1018,-27194,-1332
C00982=990,31012,-29901,1090,-27194,-1137
C00983=1210,31300,-29552,1055,-27303,-1220
C00984=1418,31602,-29186,1021,-27416,-1298
C00985=1418,31602,-27786,1021,-27416,-1298
C00986=1367,31493,-25318,1030,-27376,-1279
C00987=1367,31493,-29318,1030,-27376,-1279
C00988=1369,31486,-29327,1029,-27373,-1280
C00989=1351,31483,-29330,1032,-27372,-1273
C00990=1334,31481,-29333,1035,-27371,-1266
C00991=1316,31478,-29336,1037,-27370,-1259
C00992=1298,31476,-29340,1040,-27369,-1253
C00993=1281,31473,-29343,1042,-27367,-1246
C00994=1263,31470,-29346,1045,-27366,-1239
C00995=1245,31468,-29349,1047,-27365,-1232
C00996=1230,31460,-29359,1050,-27362,-1226
C00997=1215,31454,-29367,1052,-27360,-1220
C00998=1197,31451,-29370,1055,-27359,-1213
C00999=1179,31449,-29373,1057,-27357,-1206
C01000=1161,31446,-29376,1060,-27356,-1200
C01001=1144,31444,-29380,1062,-27355,-1193
C01002=1126,31441,-29383,1065,-27354,-1186
C01003=1112,31448,-29374,1067,-27357,-1180
C01004=1094,31446,-29377,1069,-27355,-1173
C01005=1076,31443,-29380,1072,-27354,-1166
C01006=1059,31441,-29384,1074,-27353,-1160
C01007=1041,31438,-29387,1077,-27352,-1153
C01008=1023,31436,-29390,1080,-27351,-1146
C01009=1006,31433,-29393,1082,-27350,-1139
C01010=988,31430,-29396,1085,-27349,-1132
C01011=970,31428,-29400,1087,-27348,-1125
C01012=953,31425,-29403,1090,-27346,-1118
C01013=935,31423,-29406,1092,-27345,-1112
C01014=917,31420,-29409,1095,-27344,-1105
C01015=899,31417,-29413,1098,-27343,-1098
C01016=882,31415,-29416,1100,-27342,-1091
C01017=864,31412,-29419,1103,-27341,-1084
C01018=855,31420,-29410,1104,-27343,-1080
C01019=872,31423,-29406,1102,-27345,-1087
C01020=889,31426,-29403,1099,-27346,-1094
C01021=907,31428,-29400,1096,-27347,-1101
C01022=925,31431,-29396,1094,-27348,-1108
C01023=943,31433,-29393,1091,-27349,-1114
C01024=960,31436,-29390,1089,-27350,-1121
C01025=978,31438,-29387,1086,-27352,-1128
C01026=996,31441,-29384,1084,-27353,-1135
C01027=1013,31444,-29380,1081,-27354,-1142
C01028=1031,31446,-29377,1078,-27355,-1149
C01029=1049,31449,-29374,1076,-27356,-1156
C01030=1066,31451,-29371,1073,-27357,-1162
C01031=1084,31454,-29367,1071,-27358,-1169
C01032=1102,31457,-29364,1068,-27359,-1176
C01033=1120,31459,-29361,1066,-27361,-1183
C01034=1137,31462,-29358,1063,-27362,-1190
C01035=1155,31464,-29354,1060,-27363,-1197
C01036=1173,31467,-29351,1058,-27364,-1204
C01037=1190,31469,-29348,1055,-27365,-1211
C01038=1208,31472,-29345,1053,-27366,-1217
C01039=1226,31475,-29341,1050,-27367,-1224
C01040=1243,31477,-29338,1048,-27369,-1231
C01041=1261,31480,-29335,1045,-27370,-1238
C01042=1279,31482,-29332,1042,-27371,-1245
C01043=1297,31485,-29328,1040,-27372,-1252
C01044=1314,31487,-29325,1037,-27373,-1259
C01045=1332,31490,-29322,1035,-27374,-1265
C01046=1350,31493,-29319,1032,-27375,-1272
C01047=1367,31493,-27918,1030,-27376,-1279
C01048=-41004,59868,4099,4900,-34257,16705
C01049=-41004,59868,1099,4900,-34257,16705
C01050=-41004,64596,1380,5213,-31659,16463
C01051=-41004,59868,1099,4900,-34257,16705
C01052=-41004,59868,9099,4900,-34257,16705
C01053=1367,31493,-25318,1030,-27376,-1279
C01054=1367,31493,-29318,1030,-27376,-1279
C01055=1367,31493,-27918,1030,-27376,-1279
C01056=1850,31497,-25310,960,-27382,-1467
C01057=1850,31497,-29310,960,-27382,-1467
C01058=1848,31523,-29278,960,-27392,-1466
C01059=1857,31528,-29272,959,-27394,-1470
C01060=1869,31507,-29297,957,-27386,-1474
C01061=1871,31481,-29329,957,-27376,-1475
C01062=1883,31460,-29354,956,-27369,-1480
C01063=1885,31434,-29386,956,-27359,-1481
C01064=1887,31408,-29417,956,-27349,-1482
C01065=1899,31387,-29443,954,-27342,-1487
C01066=1909,31365,-29469,953,-27334,-1491
C01067=1916,31342,-29497,952,-27325,-1494
C01068=1924,31319,-29525,952,-27317,-1497
C01069=1936,31298,-29550,950,-27309,-1502
C01070=1945,31276,-29577,949,-27301,-1506
C01071=1953,31253,-29605,948,-27293,-1509
C01072=1962,31230,-29632,947,-27284,-1513
C01073=1973,31209,-29657,946,-27277,-1517
C01074=1985,31188,-29682,944,-27269,-1522
C01075=1996,31167,-29708,943,-27261,-1526
C01076=2004,31144,-29736,942,-27253,-1530
C01077=2011,31120,-29764,941,-27244,-1533
C01078=2023,31099,-29789,940,-27237,-1537
C01079=2035,31078,-29814,938,-27229,-1542
C01080=2046,31058,-29840,937,-27221,-1547
C01081=2058,31037,-29865,935,-27214,-1552
C01082=2069,31015,-29891,934,-27206,-1556
C01083=2082,30995,-29915,932,-27199,-1561
C01084=2094,30974,-29940,931,-27191,-1566
C01085=2106,30953,-29965,930,-27183,-1571
C01086=2120,30934,-29989,928,-27176,-1576
C01087=2139,30917,-30009,925,-27170,-1584
C01088=2156,30898,-30031,923,-27164,-1590
C01089=2141,30891,-30040,925,-27161,-1585
C01090=2127,30911,-30017,927,-27168,-1579
C01091=2108,30927,-29996,930,-27174,-1572
C01092=2096,30948,-29971,931,-27181,-1567
C01093=2084,30969,-29946,933,-27189,-1562
C01094=2069,30989,-29923,934,-27196,-1556
C01095=2055,31008,-29899,936,-27203,-1551
C01096=2041,31028,-29876,938,-27210,-1545
C01097=2033,31051,-29848,939,-27219,-1542
C01098=2019,31070,-29824,941,-27226,-1536
C01099=2011,31094,-29796,942,-27234,-1533
C01100=2001,31115,-29770,943,-27242,-1529
C01101=1989,31136,-29745,944,-27250,-1524
C01102=1982,31160,-29717,945,-27259,-1521
C01103=1968,31179,-29693,947,-27266,-1515
C01104=1960,31202,-29665,948,-27274,-1512
C01105=1952,31225,-29638,949,-27282,-1509
C01106=1940,31246,-29613,950,-27290,-1504
C01107=1928,31267,-29588,952,-27298,-1499
C01108=1917,31288,-29562,953,-27305,-1495
C01109=1914,31314,-29531,953,-27315,-1494
C01110=1903,31335,-29506,954,-27323,-1489
C01111=1891,31356,-29480,956,-27330,-1484
C01112=1887,31381,-29450,956,-27340,-1483
C01113=1877,31403,-29424,957,-27347,-1478
C01114=1873,31428,-29393,958,-27357,-1476
C01115=1863,31450,-29367,959,-27365,-1473
C01116=1861,31476,-29335,959,-27374,-1472
C01117=1850,31497,-29310,960,-27382,-1467
C01118=1850,31497,-27910,960,-27382,-1467
C01119=2067,31186,-25684,933,-27269,-1554
C01120=2067,31186,-29684,933,-27269,-1554
C01121=2078,31171,-29702,931,-27264,-1558
C01122=2089,31156,-29720,930,-27258,-1563
C01123=2101,31141,-29738,928,-27253,-1567
C01124=2112,31126,-29756,927,-27247,-1572
C01125=2114,31106,-29780,927,-27240,-1573
C01126=2125,31091,-29798,925,-27235,-1577
C01127=2137,31076,-29816,924,-27229,-1582
C01128=2150,31063,-29833,922,-27224,-1587
C01129=2160,31047,-29852,921,-27218,-1591
C01130=2171,31032,-29870,919,-27213,-1595
C01131=2182,31017,-29888,918,-27208,-1600
C01132=2195,31003,-29905,916,-27202,-1605
C01133=2205,30987,-29924,915,-27197,-1609
C01134=2216,30972,-29942,913,-27191,-1614
C01135=2228,30957,-29960,912,-27186,-1618
C01136=2239,30942,-29978,910,-27181,-1623
C01137=2250,30927,-29996,909,-27175,-1627
C01138=2260,30911,-30016,908,-27169,-1631
C01139=2269,30895,-30035,907,-27163,-1635
C01140=2279,30879,-30054,905,-27158,-1638
C01141=2288,30863,-30073,904,-27152,-1642
C01142=2305,30851,-30088,902,-27147,-1649
C01143=2315,30835,-30107,901,-27142,-1653
C01144=2331,30823,-30121,898,-27137,-1659
C01145=2348,30811,-30136,896,-27133,-1666
C01146=2364,30799,-30151,894,-27129,-1672
C01147=2374,30783,-30170,893,-27123,-1676
C01148=2390,30771,-30184,890,-27118,-1683
C01149=2400,30755,-30203,889,-27113,-1686
C01150=2410,30739,-30223,888,-27107,-1690
C01151=2393,30751,-30208,890,-27111,-1684
C01152=2377,30763,-30193,892,-27116,-1677
C01153=2360,30775,-30179,895,-27120,-1671
C01154=2350,30791,-30160,896,-27126,-1667
C01155=2334,30803,-30145,898,-27130,-1660
C01156=2317,30815,-30131,900,-27134,-1654
C01157=2301,30827,-30116,903,-27139,-1647
C01158=2291,30843,-30097,904,-27144,-1643
C01159=2277,30857,-30081,906,-27149,-1638
C01160=2265,30871,-30063,907,-27155,-1633
C01161=2254,30887,-30045,909,-27160,-1629
C01162=2243,30902,-30027,910,-27166,-1624
C01163=2231,30917,-30009,912,-27171,-1620
C01164=2220,30931,-29991,913,-27176,-1615
C01165=2210,30947,-29972,915,-27182,-1611
C01166=2200,30963,-29953,916,-27188,-1607
C01167=2191,30979,-29934,917,-27194,-1604
C01168=2181,30995,-29914,918,-27200,-1600
C01169=2165,31007,-29900,920,-27204,-1593
C01170=2155,31023,-29881,922,-27210,-1589
C01171=2146,31039,-29862,923,-27215,-1586
C01172=2136,31055,-29842,924,-27221,-1582
C01173=2127,31071,-29823,925,-27227,-1578
C01174=2115,31086,-29805,927,-27233,-1573
C01175=2104,31101,-29787,928,-27238,-1569
C01176=2093,31116,-29769,930,-27243,-1564
C01177=2088,31135,-29746,930,-27250,-1563
C01178=2080,31151,-29727,931,-27256,-1559
C01179=2069,31166,-29708,932,-27262,-1555
C01180=2067,31186,-29684,933,-27269,-1554
C01181=2067,31186,-28284,933,-27269,-1554
C01182=2241,31045,-25853,909,-27219,-1623
C01183=2241,31045,-29853,909,-27219,-1623
C01184=2246,31045,-29854,908,-27219,-1625
C01185=2255,31039,-29861,907,-27216,-1628
C01186=2263,31032,-29869,906,-27214,-1631
C01187=2265,31022,-29881,906,-27210,-1632
C01188=2273,31016,-29888,905,-27208,-1635
C01189=2275,31006,-29900,904,-27205,-1636
C01190=2276,30996,-29912,904,-27201,-1637
C01191=2285,30990,-29920,903,-27199,-1640
C01192=2287,30980,-29931,903,-27195,-1641
C01193=2295,30974,-29939,902,-27193,-1644
C01194=2299,30965,-29950,901,-27190,-1646
C01195=2305,30957,-29959,901,-27187,-1648
C01196=2310,30949,-29969,900,-27184,-1650
C01197=2315,30941,-29979,899,-27181,-1652
C01198=2322,30934,-29987,898,-27178,-1655
C01199=2325,30925,-29998,898,-27175,-1656
C01200=2333,30919,-30006,897,-27173,-1659
C01201=2335,30909,-30018,897,-27169,-1660
C01202=2344,30902,-30025,896,-27167,-1663
C01203=2346,30893,-30037,895,-27163,-1664
C01204=2354,30886,-30045,894,-27161,-1667
C01205=2357,30877,-30056,894,-27158,-1669
C01206=2364,30870,-30064,893,-27155,-1671
C01207=2369,30862,-30074,892,-27152,-1673
C01208=2374,30854,-30084,892,-27149,-1676
C01209=2382,30848,-30091,891,-27147,-1679
C01210=2391,30841,-30099,889,-27145,-1682
C01211=2392,30831,-30111,889,-27141,-1683
C01212=2401,30825,-30118,888,-27139,-1686
C01213=2403,30815,-30130,888,-27135,-1687
C01214=2393,30813,-30133,889,-27134,-1683
C01215=2392,30823,-30121,890,-27138,-1683
C01216=2383,30829,-30114,891,-27140,-1679
C01217=2381,30839,-30102,891,-27144,-1678
C01218=2373,30845,-30094,892,-27146,-1675
C01219=2365,30852,-30087,893,-27148,-1672
C01220=2359,30859,-30077,894,-27151,-1670
C01221=2354,30868,-30067,894,-27154,-1668
C01222=2346,30874,-30059,896,-27156,-1665
C01223=2337,30880,-28652,897,-27159,-1661
C01224=-41004,59868,4099,4900,-34257,16705
C01225=-41004,59868,1099,4900,-34257,16705
C01226=-41004,64596,1380,5213,-31659,16463
C01227=-41004,59868,1099,4900,-34257,16705
C01228=-41004,59868,9099,4900,-34257,16705
C01229=2337,30880,-26052,897,-27159,-1661
C01230=2337,30880,-30052,897,-27159,-1661
C01231=2336,30890,-30040,897,-27162,-1660
C01232=2327,30897,-30032,898,-27165,-1657
C01233=2324,30906,-30021,898,-27168,-1656
C01234=2317,30913,-30013,899,-27170,-1653
C01235=2313,30921,-30003,900,-27173,-1651
C01236=2307,30929,-29993,901,-27176,-1649
C01237=2301,30937,-29984,901,-27179,-1647
C01238=2297,30945,-29974,902,-27182,-1645
C01239=2290,30952,-29966,903,-27185,-1642
C01240=2287,30962,-29954,903,-27188,-1641
C01241=2279,30968,-29947,904,-27190,-1638
C01242=2277,30978,-29934,904,-27194,-1637
C01243=2276,30988,-29922,905,-27198,-1636
C01244=2267,30994,-29915,906,-27200,-1633
C01245=2265,31004,-29903,906,-27204,-1632
C01246=2264,31014,-29891,906,-27207,-1632
C01247=2255,31020,-29883,907,-27210,-1628
C01248=2253,31030,-29872,907,-27213,-1627
C01249=2245,31037,-29864,908,-27216,-1624
C01250=2241,31045,-29853,909,-27219,-1623
C01251=2241,31045,-28453,909,-27219,-1623
C01252=2612,31005,-25899,856,-27207,-1767
C01253=2612,31005,-29899,856,-27207,-1767
C01254=2620,31017,-29886,854,-27212,-1770
C01255=2622,31029,-29870,854,-27216,-1770
C01256=2631,31040,-29857,853,-27220,-1774
C01257=2639,31051,-29844,851,-27225,-1777
C01258=2642,31063,-29829,851,-27229,-1778
C01259=2653,31071,-29820,849,-27232,-1782
C01260=2658,31062,-29831,848,-27229,-1784
C01261=2649,31051,-29844,850,-27225,-1781
C01262=2647,31038,-29859,850,-27220,-1780
C01263=2638,31028,-29872,852,-27216,-1777
C01264=2632,31016,-29886,853,-27211,-1774
C01265=2633,31003,-29902,853,-27207,-1775
C01266=2625,30992,-29916,854,-27202,-1772
C01267=2625,30979,-29932,854,-27198,-1772
C01268=2626,30965,-29948,854,-27193,-1773
C01269=2627,30952,-29964,854,-27188,-1773
C01270=2628,30939,-29980,854,-27183,-1774
C01271=2629,30926,-29996,854,-27178,-1774
C01272=2630,30912,-30012,854,-27173,-1775
C01273=2632,30899,-30028,854,-27168,-1775
C01274=2633,30886,-30044,854,-27163,-1776
C01275=2644,30878,-30053,852,-27160,-1780
C01276=2648,30866,-30067,852,-27156,-1782
C01277=2660,30861,-30073,850,-27154,-1786
C01278=2672,30857,-30078,849,-27153,-1791
C01279=2683,30849,-30087,847,-27150,-1796
C01280=2694,30842,-30097,846,-27147,-1800
C01281=2705,30834,-30106,844,-27145,-1804
C01282=2710,30823,-30120,843,-27141,-1806
C01283=2720,30814,-30130,842,-27137,-1810
C01284=2730,30806,-30140,841,-27135,-1814
C01285=2741,30798,-30149,839,-27132,-1819
C01286=2745,30786,-30163,839,-27127,-1820
C01287=2755,30778,-30174,837,-27124,-1824
C01288=2756,30764,-30190,837,-27119,-1825
C01289=2746,30759,-30196,839,-27117,-1821
C01290=2742,30771,-30182,839,-27122,-1819
C01291=2732,30779,-30173,841,-27125,-1815
C01292=2723,30788,-30161,842,-27128,-1812
C01293=2717,30798,-30149,843,-27132,-1809
C01294=2706,30806,-30139,844,-27135,-1805
C01295=2700,30817,-30126,845,-27139,-1802
C01296=2691,30826,-30116,846,-27142,-1799
C01297=2680,30834,-30106,848,-27144,-1794
C01298=2669,30842,-30097,849,-27147,-1790
C01299=2658,30850,-30087,851,-27150,-1786
C01300=2647,30858,-30078,852,-27153,-1782
C01301=2634,30859,-30077,854,-27153,-1776
C01302=2624,30867,-30066,855,-27156,-1773
C01303=2623,30880,-30050,855,-27161,-1772
C01304=2615,30890,-30039,856,-27165,-1769
C01305=2611,30902,-30025,857,-27169,-1767
C01306=2610,30915,-30009,857,-27174,-1767
C01307=2609,30928,-29993,857,-27179,-1766
C01308=2607,30941,-29977,857,-27184,-1766
C01309=2606,30955,-29961,857,-27189,-1765
C01310=2605,30968,-29945,857,-27193,-1764
C01311=2614,30979,-29931,856,-27198,-1768
C01312=2613,30992,-29915,856,-27202,-1767
C01313=2612,31005,-29899,856,-27207,-1767
C01314=2612,31005,-28499,856,-27207,-1767
C01315=2556,30880,-26052,865,-27160,-1746
C01316=2556,30880,-30052,865,-27160,-1746
C01317=2565,30844,-30094,864,-27147,-1750
C01318=2578,30811,-30134,863,-27135,-1755
C01319=2602,30786,-30165,859,-27126,-1765
C01320=2636,30769,-30185,855,-27120,-1778
C01321=2660,30742,-30217,851,-27110,-1787
C01322=2687,30722,-30242,848,-27103,-1798
C01323=2721,30707,-30259,843,-27098,-1811
C01324=2755,30691,-30278,838,-27092,-1824
C01325=2786,30669,-30305,834,-27084,-1837
C01326=2818,30646,-30333,830,-27076,-1849
C01327=2835,30615,-30370,827,-27065,-1856
C01328=2854,30586,-30405,825,-27054,-1864
C01329=2865,30554,-30444,824,-27042,-1868
C01330=2861,30517,-30488,825,-27029,-1867
C01331=2849,30483,-30530,827,-27016,-1862
C01332=2844,30446,-30574,828,-27002,-1861
C01333=2839,30410,-30618,829,-26989,-1859
C01334=2843,30372,-30664,829,-26975,-1861
C01335=2856,30339,-30704,827,-26963,-1866
C01336=2878,30311,-30738,824,-26952,-1875
C01337=2903,30284,-30770,821,-26943,-1885
C01338=2926,30257,-30803,818,-26933,-1894
C01339=2938,30223,-30843,816,-26921,-1899
C01340=2942,30186,-30889,816,-26907,-1901
C01341=2956,30153,-30928,815,-26895,-1906
C01342=2959,30115,-30974,814,-26880,-1908
C01343=2963,30076,-31021,814,-26866,-1909
C01344=2966,30038,-31067,814,-26852,-1911
C01345=2982,30007,-31105,812,-26841,-1917
C01346=2971,29988,-31127,814,-26834,-1913
C01347=2957,30021,-31087,816,-26846,-1908
C01348=2944,30054,-31048,817,-26858,-1902
C01349=2941,30092,-31001,817,-26872,-1901
C01350=2937,30130,-30955,818,-26886,-1899
C01351=2944,30166,-30912,816,-26899,-1902
C01352=2926,30197,-30875,818,-26911,-1895
C01353=2909,30227,-30839,821,-26922,-1887
C01354=2894,30259,-30800,822,-26934,-1882
C01355=2871,30287,-30767,826,-26943,-1873
C01356=2849,30314,-30733,829,-26954,-1864
C01357=2835,30347,-30694,830,-26965,-1858
C01358=2821,30380,-30654,832,-26978,-1853
C01359=2818,30418,-30608,832,-26992,-1851
C01360=2825,30454,-30565,831,-27005,-1854
C01361=2832,30490,-30522,829,-27018,-1856
C01362=2840,30525,-30479,828,-27032,-1859
C01363=2846,30561,-30435,826,-27045,-1861
C01364=2833,30594,-30395,828,-27057,-1856
C01365=2820,30627,-30356,830,-27069,-1850
C01366=2795,30653,-30324,833,-27079,-1840
C01367=2761,30669,-30305,838,-27084,-1827
C01368=2727,30685,-30286,842,-27090,-1814
C01369=2691,30694,-30276,847,-27093,-1800
C01370=2658,30709,-30257,852,-27098,-1787
C01371=2640,30739,-30221,854,-27109,-1780
C01372=2609,30762,-30193,859,-27117,-1767
C01373=2577,30785,-30166,863,-27125,-1755
C01374=2557,30814,-30131,866,-27136,-1747
C01375=2554,30852,-30085,866,-27150,-1745
C01376=2556,30880,-30052,865,-27160,-1746
C01377=2556,30880,-28652,865,-27160,-1746
C01378=2589,30685,-26287,862,-27089,-1760
C01379=2589,30685,-30287,862,-27089,-1760
C01380=2594,30684,-30287,862,-27088,-1762
C01381=2600,30677,-30296,861,-27086,-1764
C01382=2601,30667,-30309,861,-27082,-1765
C01383=2605,30659,-30318,860,-27079,-1767
C01384=2612,30652,-30326,859,-27077,-1769
C01385=2613,30642,-30338,859,-27073,-1770
C01386=2616,30633,-30349,859,-27070,-1771
C01387=2624,30627,-30357,858,-27067,-1774
C01388=2625,30617,-30368,858,-27064,-1775
C01389=2626,30607,-30381,858,-27060,-1775
C01390=2627,30597,-30393,858,-27056,-1776
C01391=2628,30587,-30405,858,-27053,-1776
C01392=2631,30578,-30416,857,-27049,-1777
C01393=2639,30572,-30423,856,-27047,-1781
C01394=2640,30562,-30435,856,-27043,-1781
C01395=2642,30552,-30447,856,-27040,-1782
C01396=2650,30546,-30454,855,-27038,-1785
C01397=2653,30537,-30465,855,-27034,-1786
C01398=2660,30530,-30473,854,-27032,-1789
C01399=2665,30523,-29083,853,-27029,-1791
C01400=-41004,59868,4099,4900,-34257,16705
C01401=-41004,59868,1099,4900,-34257,16705
C01402=-41004,64596,1380,5213,-31659,16463
C01403=-41004,59868,1099,4900,-34257,16705
C01404=-41004,59868,9099,4900,-34257,16705
C01405=2665,30523,-26483,853,-27029,-1791
C01406=2665,30523,-30483,853,-27029,-1791
C01407=2669,30515,-30492,853,-27026,-1793
C01408=2676,30508,-30500,852,-27024,-1795
C01409=2679,30499,-30511,851,-27020,-1797
C01410=2687,30493,-30519,850,-27018,-1800
C01411=2689,30483,-30530,850,-27015,-1800
C01412=2697,30477,-30538,849,-27012,-1804
C01413=2700,30468,-30548,849,-27009,-1805
C01414=2701,30458,-30560,849,-27005,-1805
C01415=2702,30448,-30573,849,-27002,-1806
C01416=2703,30438,-30585,849,-26998,-1806
C01417=2693,30436,-30587,850,-26997,-1802
C01418=2692,30446,-30575,850,-27001,-1802
C01419=2690,30455,-30564,850,-27004,-1801
C01420=2682,30461,-30556,851,-27007,-1798
C01421=2679,30471,-30545,852,-27010,-1797
C01422=2678,30481,-30533,852,-27014,-1796
C01423=2671,30487,-30525,853,-27016,-1793
C01424=2667,30496,-30515,853,-27019,-1792
C01425=2661,30503,-30506,854,-27022,-1790
C01426=2655,30510,-30497,855,-27024,-1787
C01427=2651,30519,-30487,855,-27028,-1786
C01428=2644,30525,-30480,856,-27030,-1783
C01429=2642,30535,-30468,856,-27033,-1782
C01430=2633,30541,-30461,858,-27035,-1779
C01431=2631,30550,-30450,858,-27039,-1778
C01432=2624,30556,-30442,859,-27041,-1775
C01433=2620,30565,-30432,859,-27044,-1773
C01434=2619,30575,-30420,859,-27048,-1773
C01435=2618,30585,-30408,859,-27052,-1772
C01436=2617,30595,-30395,859,-27055,-1772
C01437=2616,30605,-30383,859,-27059,-1771
C01438=2609,30612,-30375,860,-27062,-1769
C01439=2605,30620,-30365,861,-27065,-1767
C01440=2604,30630,-30353,861,-27068,-1766
C01441=2603,30640,-30341,861,-27072,-1766
C01442=2602,30650,-30329,861,-27076,-1766
C01443=2595,30657,-30321,862,-27078,-1763
C01444=2590,30665,-30311,862,-27081,-1761
C01445=2590,30675,-30299,862,-27085,-1761
C01446=2589,30685,-30287,862,-27089,-1760
C01447=2589,30685,-28887,862,-27089,-1760
C01448=2654,30638,-26343,853,-27072,-1786
C01449=2654,30638,-30343,853,-27072,-1786
C01450=2657,30638,-30343,853,-27072,-1787
C01451=2662,30635,-30347,852,-27071,-1789
C01452=2667,30631,-30351,852,-27069,-1791
C01453=2672,30628,-30355,851,-27068,-1793
C01454=2676,30624,-30360,850,-27067,-1795
C01455=2681,30621,-30364,850,-27066,-1797
C01456=2686,30617,-30368,849,-27064,-1798
C01457=2692,30617,-30368,848,-27064,-1801
C01458=2698,30617,-30368,847,-27064,-1803
C01459=2703,30614,-30372,847,-27063,-1805
C01460=2708,30610,-30376,846,-27062,-1807
C01461=2713,30607,-30380,845,-27061,-1809
C01462=2718,30603,-30385,845,-27059,-1811
C01463=2723,30600,-30389,844,-27058,-1813
C01464=2727,30596,-30393,843,-27057,-1815
C01465=2732,30593,-30397,843,-27056,-1816
C01466=2737,30589,-30402,842,-27054,-1818
C01467=2742,30586,-30406,841,-27053,-1820
C01468=2747,30582,-30410,841,-27052,-1822
C01469=2752,30579,-30414,840,-27051,-1824
C01470=2753,30573,-30421,840,-27049,-1825
C01471=2754,30568,-30427,840,-27047,-1825
C01472=2759,30564,-30432,839,-27045,-1827
C01473=2764,30561,-30436,838,-27044,-1829
C01474=2765,30555,-30443,838,-27042,-1829
C01475=2765,30549,-30450,838,-27040,-1830
C01476=2766,30543,-30457,838,-27038,-1830
C01477=2766,30537,-30464,838,-27035,-1830
C01478=2767,30531,-30471,838,-27033,-1830
C01479=2767,30525,-30479,838,-27031,-1831
C01480=2764,30523,-30482,839,-27030,-1829
C01481=2757,30522,-30483,840,-27030,-1827
C01482=2757,30528,-30476,840,-27032,-1826
C01483=2754,30532,-30470,840,-27034,-1826
C01484=2750,30536,-30466,841,-27035,-1824
C01485=2745,30540,-30461,841,-27036,-1822
C01486=2745,30546,-30454,841,-27038,-1822
C01487=2744,30552,-30447,841,-27041,-1821
C01488=2744,30558,-30440,841,-27043,-1821
C01489=2739,30561,-30436,842,-27044,-1819
C01490=2734,30565,-30431,843,-27045,-1818
C01491=2730,30568,-30427,843,-27047,-1816
C01492=2725,30572,-30423,844,-27048,-1814
C01493=2720,30575,-30419,845,-27049,-1812
C01494=2715,30579,-30414,845,-27050,-1810
C01495=2710,30582,-30410,846,-27052,-1808
C01496=2705,30586,-30406,847,-27053,-1806
C01497=2700,30589,-30402,847,-27054,-1804
C01498=2696,30593,-30398,848,-27055,-1802
C01499=2691,30596,-30393,849,-27057,-1800
C01500=2686,30600,-30389,849,-27058,-1798
C01501=2681,30603,-30385,850,-27059,-1797
C01502=2676,30607,-30381,851,-27060,-1795
C01503=2671,30610,-30376,851,-27062,-1793
C01504=2666,30614,-30372,852,-27063,-1791
C01505=2662,30617,-30368,853,-27064,-1789
C01506=2657,30621,-30364,853,-27065,-1787
C01507=2655,30626,-30357,853,-27067,-1786
C01508=2655,30632,-30350,853,-27070,-1786
C01509=2654,30638,-30343,853,-27072,-1786
C01510=2654,30638,-28943,853,-27072,-1786
C01511=2364,30453,-26569,898,-27001,-1675
C01512=2364,30453,-30569,898,-27001,-1675
C01513=2372,30447,-30576,896,-26998,-1678
C01514=2374,30437,-30588,896,-26995,-1679
C01515=2382,30431,-30595,895,-26993,-1682
C01516=2385,30423,-30605,895,-26990,-1683
C01517=2391,30416,-30613,894,-26987,-1685
C01518=2396,30408,-30622,893,-26984,-1688
C01519=2397,30399,-30634,893,-26981,-1688
C01520=2398,30389,-30646,893,-26977,-1688
C01521=2399,30379,-30658,893,-26974,-1689
C01522=2400,30369,-30670,893,-26970,-1689
C01523=2400,30359,-30681,893,-26966,-1690
C01524=2401,30350,-30693,893,-26963,-1690
C01525=2402,30340,-30705,893,-26959,-1690
C01526=2403,30330,-30717,893,-26955,-1691
C01527=2404,30320,-30729,893,-26952,-1691
C01528=2404,30310,-30741,893,-26948,-1691
C01529=2399,30302,-30751,894,-26945,-1690
C01530=2396,30293,-30762,895,-26942,-1688
C01531=2396,30283,-30773,895,-26938,-1689
C01532=2397,30273,-30785,895,-26935,-1689
C01533=2398,30264,-30797,895,-26931,-1689
C01534=2394,30255,-30808,895,-26928,-1688
C01535=2389,30246,-30818,896,-26924,-1686
C01536=2390,30237,-30830,896,-26921,-1686
C01537=2389,30227,-30841,897,-26917,-1686
C01538=2382,30219,-30851,898,-26914,-1683
C01539=2382,30210,-30863,898,-26911,-1683
C01540=2372,30208,-30865,899,-26910,-1680
C01541=2371,30217,-30853,899,-26914,-1679
C01542=2370,30227,-30841,899,-26917,-1679
C01543=2370,30237,-30829,899,-26921,-1679
C01544=2377,30245,-30820,898,-26924,-1681
C01545=2378,30254,-30808,898,-26927,-1682
C01546=2377,30264,-30797,898,-26931,-1681
C01547=2377,30274,-30785,898,-26935,-1681
C01548=2376,30284,-30773,898,-26938,-1681
C01549=2382,30292,-30763,897,-26941,-1683
C01550=2385,30301,-30752,896,-26945,-1684
C01551=2384,30311,-30740,896,-26948,-1683
C01552=2383,30321,-30728,896,-26952,-1683
C01553=2382,30330,-30716,896,-26956,-1683
C01554=2381,30340,-30705,896,-26959,-1682
C01555=2381,30350,-30693,896,-26963,-1682
C01556=2380,30360,-30681,896,-26966,-1682
C01557=2379,30370,-30669,896,-26970,-1681
C01558=2378,30380,-30657,896,-26974,-1681
C01559=2377,30389,-30645,896,-26977,-1680
C01560=2376,30399,-30633,896,-26981,-1680
C01561=2376,30409,-30621,896,-26985,-1680
C01562=2368,30415,-30614,898,-26987,-1676
C01563=2364,30423,-30604,898,-26990,-1675
C01564=2363,30433,-30592,898,-26993,-1675
C01565=2357,30440,-30584,899,-26996,-1672
C01566=2352,30447,-30575,899,-26998,-1670
C01567=2348,30456,-30565,900,-27002,-1669
C01568=2340,30462,-30558,901,-27004,-1665
C01569=2340,30470,-30548,901,-27007,-1665
C01570=2348,30464,-30555,900,-27005,-1669
C01571=2356,30458,-30562,899,-27003,-1672
C01572=2364,30453,-29169,898,-27001,-1675
C01573=-41004,59868,4099,4900,-34257,16705
C01574=-41004,59868,1099,4900,-34257,16705
C01575=-41004,64596,1380,5213,-31659,16463
C01576=-41004,59868,1099,4900,-34257,16705
C01577=-41004,59868,9099,4900,-34257,16705
C01578=2364,30453,-26569,898,-27001,-1675
C01579=2364,30453,-30569,898,-27001,-1675
C01580=2364,30453,-29169,898,-27001,-1675
C01581=2523,30248,-26815,877,-26926,-1738
C01582=2523,30248,-30815,877,-26926,-1738
C01583=2529,30245,-30819,876,-26925,-1740
C01584=2534,30241,-30824,875,-26924,-1742
C01585=2540,30236,-30829,874,-26922,-1745
C01586=2546,30232,-30834,874,-26921,-1747
C01587=2552,30228,-30839,873,-26919,-1749
C01588=2555,30224,-30845,872,-26917,-1751
C01589=2550,30218,-30852,873,-26915,-1749
C01590=2547,30212,-30859,874,-26913,-1747
C01591=2548,30205,-30867,874,-26910,-1748
C01592=2548,30198,-30876,874,-26908,-1748
C01593=2549,30191,-30884,874,-26905,-1748
C01594=2549,30184,-30893,874,-26903,-1749
C01595=2550,30177,-30901,874,-26900,-1749
C01596=2546,30171,-30908,874,-26898,-1747
C01597=2541,30165,-30915,875,-26896,-1745
C01598=2541,30158,-30924,875,-26893,-1746
C01599=2542,30151,-30932,875,-26891,-1746
C01600=2541,30145,-30940,875,-26888,-1746
C01601=2536,30139,-30947,876,-26886,-1744
C01602=2530,30135,-30952,877,-26884,-1741
C01603=2523,30134,-30953,878,-26884,-1739
C01604=2518,30128,-30960,879,-26882,-1737
C01605=2512,30123,-30967,880,-26880,-1735
C01606=2505,30122,-30968,881,-26879,-1732
C01607=2497,30121,-30969,882,-26879,-1729
C01608=2490,30120,-30971,883,-26878,-1726
C01609=2482,30119,-30972,884,-26878,-1723
C01610=2475,30117,-30973,885,-26877,-1720
C01611=2467,30116,-30975,886,-26877,-1717
C01612=2459,30115,-30976,887,-26877,-1714
C01613=2452,30114,-30977,889,-26876,-1711
C01614=2451,30121,-30969,889,-26879,-1711
C01615=2451,30128,-30961,889,-26881,-1711
C01616=2450,30135,-30952,889,-26884,-1710
C01617=2450,30142,-30944,889,-26886,-1710
C01618=2457,30143,-30942,888,-26887,-1713
C01619=2463,30141,-30944,887,-26886,-1715
C01620=2469,30137,-30949,886,-26885,-1718
C01621=2476,30137,-30950,885,-26885,-1720
C01622=2483,30138,-30949,884,-26885,-1723
C01623=2491,30139,-30947,883,-26886,-1726
C01624=2496,30145,-30941,882,-26888,-1728
C01625=2501,30150,-30934,881,-26890,-1730
C01626=2509,30151,-30933,880,-26890,-1733
C01627=2514,30155,-30927,879,-26892,-1735
C01628=2519,30161,-30920,878,-26894,-1737
C01629=2524,30167,-30913,877,-26896,-1739
C01630=2529,30173,-30906,877,-26898,-1741
C01631=2529,30179,-30898,877,-26901,-1741
C01632=2529,30186,-30890,877,-26903,-1740
C01633=2529,30193,-30882,876,-26906,-1741
C01634=2534,30199,-30875,876,-26908,-1742
C01635=2537,30205,-30867,875,-26910,-1744
C01636=2537,30212,-30859,875,-26913,-1743
C01637=2536,30219,-30850,875,-26916,-1743
C01638=2533,30224,-30844,876,-26917,-1742
C01639=2527,30228,-30839,876,-26919,-1739
C01640=2524,30234,-30832,877,-26921,-1739
C01641=2524,30241,-30823,877,-26924,-1738
C01642=2523,30248,-30815,877,-26926,-1738
C01643=2523,30248,-29415,877,-26926,-1738
C01644=2408,30154,-26929,894,-26891,-1694
C01645=2408,30154,-30929,894,-26891,-1694
C01646=2413,30151,-30933,894,-26889,-1696
C01647=2417,30148,-30937,893,-26888,-1698
C01648=2418,30143,-30942,893,-26887,-1698
C01649=2419,30138,-30949,893,-26885,-1698
C01650=2419,30133,-30955,893,-26883,-1699
C01651=2420,30127,-30961,893,-26881,-1699
C01652=2420,30122,-30968,893,-26879,-1699
C01653=2419,30117,-30974,893,-26877,-1699
C01654=2415,30113,-30979,894,-26875,-1697
C01655=2411,30109,-30984,895,-26874,-1696
C01656=2411,30103,-30991,895,-26872,-1696
C01657=2412,30098,-30997,895,-26870,-1696
C01658=2412,30093,-31003,895,-26868,-1696
C01659=2411,30088,-31009,895,-26866,-1696
C01660=2408,30084,-31015,895,-26864,-1694
C01661=2404,30079,-31020,896,-26863,-1693
C01662=2404,30074,-31026,896,-26861,-1693
C01663=2404,30069,-31032,896,-26859,-1693
C01664=2400,30065,-31038,897,-26857,-1692
C01665=2396,30060,-31043,897,-26856,-1690
C01666=2395,30056,-31049,898,-26854,-1690
C01667=2395,30050,-31055,898,-26852,-1690
C01668=2391,30048,-31058,898,-26851,-1688
C01669=2386,30047,-31059,899,-26851,-1686
C01670=2382,30043,-31063,900,-26849,-1685
C01671=2378,30039,-31069,900,-26848,-1683
C01672=2374,30036,-31072,901,-26846,-1682
C01673=2368,30035,-31073,902,-26846,-1679
C01674=2362,30034,-31074,903,-26846,-1677
C01675=2356,30033,-31076,903,-26845,-1675
C01676=2351,30033,-31077,904,-26845,-1673
C01677=2345,30032,-31078,905,-26845,-1670
C01678=2344,30037,-31071,905,-26847,-1670
C01679=2344,30042,-31065,905,-26849,-1670
C01680=2344,30048,-31058,905,-26851,-1670
C01681=2345,30052,-31053,905,-26852,-1670
C01682=2349,30057,-31047,904,-26854,-1672
C01683=2352,30061,-31042,904,-26856,-1673
C01684=2356,30065,-31037,903,-26857,-1675
C01685=2360,30070,-31032,903,-26859,-1676
C01686=2364,30074,-31026,902,-26861,-1677
C01687=2367,30078,-31021,901,-26862,-1679
C01688=2371,30083,-31016,901,-26864,-1680
C01689=2371,30088,-31010,901,-26866,-1680
C01690=2371,30093,-31003,901,-26868,-1680
C01691=2375,30097,-30998,900,-26869,-1682
C01692=2379,30102,-30993,899,-26871,-1683
C01693=2380,30107,-30987,899,-26873,-1684
C01694=2380,30112,-30981,899,-26875,-1683
C01695=2382,30116,-30975,899,-26876,-1684
C01696=2386,30121,-30970,898,-26878,-1686
C01697=2389,30125,-30964,898,-26880,-1687
C01698=2388,30130,-30958,898,-26882,-1687
C01699=2390,30135,-30952,897,-26883,-1687
C01700=2394,30140,-30947,897,-26885,-1689
C01701=2397,30144,-30942,896,-26887,-1690
C01702=2397,30149,-30935,896,-26889,-1690
C01703=2397,30154,-30930,896,-26890,-1690
C01704=2403,30155,-30928,895,-26891,-1692
C01705=2408,30154,-30929,894,-26891,-1694
C01706=2408,30154,-29529,894,-26891,-1694
C01707=2290,30072,-27029,913,-26859,-1649
C01708=2290,30072,-31029,913,-26859,-1649
C01709=2294,30068,-31034,912,-26858,-1651
C01710=2299,30065,-31038,911,-26857,-1653
C01711=2301,30059,-31044,911,-26855,-1653
C01712=2302,30053,-31052,911,-26852,-1654
C01713=2302,30047,-31059,911,-26850,-1654
C01714=2305,30043,-31064,911,-26848,-1655
C01715=2310,30039,-31069,910,-26847,-1657
C01716=2311,30036,-31072,910,-26846,-1657
C01717=2305,30035,-31073,911,-26846,-1655
C01718=2298,30035,-31074,912,-26845,-1652
C01719=2292,30034,-31076,913,-26845,-1650
C01720=2286,30033,-31077,914,-26845,-1647
C01721=2279,30032,-31078,915,-26844,-1645
C01722=2273,30031,-31079,916,-26844,-1642
C01723=2268,30034,-31075,916,-26845,-1641
C01724=2263,30038,-31070,917,-26846,-1639
C01725=2258,30042,-31066,918,-26848,-1637
C01726=2253,30045,-31062,918,-26849,-1635
C01727=2248,30049,-31058,919,-26850,-1633
C01728=2243,30052,-31053,920,-26851,-1631
C01729=2238,30054,-31051,921,-26852,-1629
C01730=2231,30053,-31052,922,-26852,-1626
C01731=2225,30053,-31053,922,-26851,-1624
C01732=2218,30052,-31053,923,-26851,-1621
C01733=2213,30056,-31049,924,-26853,-1619
C01734=2209,30059,-31045,925,-26854,-1617
C01735=2208,30065,-31038,925,-26856,-1617
C01736=2206,30070,-31032,925,-26858,-1616
C01737=2201,30074,-31027,926,-26859,-1614
C01738=2196,30078,-31023,926,-26860,-1612
C01739=2191,30081,-31019,927,-26862,-1610
C01740=2186,30085,-31014,928,-26863,-1609
C01741=2181,30088,-31010,928,-26864,-1607
C01742=2176,30092,-31006,929,-26866,-1605
C01743=2174,30097,-31000,929,-26867,-1604
C01744=2174,30103,-30992,929,-26870,-1604
C01745=2173,30109,-30985,929,-26872,-1603
C01746=2175,30114,-30979,929,-26874,-1604
C01747=2179,30119,-30973,928,-26876,-1606
C01748=2184,30122,-29569,928,-26877,-1607
C01749=-41004,59868,4099,4900,-34257,16705
C01750=-41004,59868,1099,4900,-34257,16705
C01751=-41004,64596,1380,5213,-31659,16463
C01752=-41004,59868,1099,4900,-34257,16705
C01753=-41004,59868,9099,4900,-34257,16705
C01754=2184,30122,-26969,928,-26877,-1607
C01755=2184,30122,-30969,928,-26877,-1607
C01756=2189,30118,-30974,927,-26875,-1609
C01757=2194,30115,-30978,926,-26874,-1611
C01758=2198,30111,-30982,926,-26873,-1613
C01759=2203,30108,-30987,925,-26872,-1615
C01760=2208,30104,-30991,924,-26870,-1617
C01761=2213,30100,-30995,924,-26869,-1619
C01762=2219,30100,-30996,923,-26869,-1621
C01763=2226,30100,-30995,922,-26869,-1624
C01764=2230,30097,-30999,921,-26868,-1626
C01765=2235,30093,-31004,920,-26867,-1628
C01766=2242,30093,-31004,920,-26867,-1630
C01767=2248,30093,-31004,919,-26867,-1632
C01768=2253,30090,-31008,918,-26865,-1634
C01769=2258,30086,-31012,917,-26864,-1636
C01770=2264,30087,-31011,916,-26864,-1639
C01771=2270,30086,-31012,915,-26864,-1641
C01772=2275,30083,-31017,915,-26863,-1643
C01773=2280,30079,-31021,914,-26862,-1645
C01774=2285,30075,-31025,913,-26860,-1647
C01775=2290,30072,-31029,913,-26859,-1649
C01776=2290,30072,-29629,913,-26859,-1649
C01777=1965,30267,-26795,958,-26929,-1521
C01778=1965,30267,-30795,958,-26929,-1521
C01779=1955,30262,-30801,959,-26927,-1518
C01780=1951,30274,-30787,960,-26931,-1516
C01781=1943,30283,-30776,961,-26934,-1513
C01782=1942,30296,-30761,961,-26939,-1512
C01783=1933,30305,-30750,962,-26942,-1509
C01784=1930,30317,-30735,962,-26947,-1507
C01785=1929,30330,-30720,962,-26951,-1507
C01786=1928,30343,-30704,962,-26956,-1506
C01787=1929,30356,-30688,962,-26961,-1507
C01788=1937,30367,-30675,961,-26965,-1510
C01789=1936,30380,-30659,961,-26970,-1509
C01790=1942,30391,-30645,960,-26974,-1511
C01791=1944,30404,-30630,959,-26979,-1512
C01792=1943,30417,-30615,959,-26984,-1512
C01793=1942,30430,-30599,959,-26988,-1511
C01794=1941,30443,-30583,959,-26993,-1511
C01795=1940,30456,-30567,959,-26998,-1510
C01796=1946,30468,-30553,958,-27002,-1512
C01797=1948,30480,-30538,958,-27007,-1513
C01798=1947,30493,-30522,958,-27012,-1513
C01799=1946,30506,-30507,958,-27017,-1512
C01800=1945,30519,-30491,958,-27021,-1512
C01801=1944,30532,-30475,958,-27026,-1511
C01802=1943,30545,-30459,958,-27031,-1511
C01803=1942,30558,-30443,958,-27036,-1510
C01804=1941,30572,-30428,958,-27041,-1510
C01805=1940,30585,-30412,958,-27046,-1509
C01806=1942,30597,-30397,957,-27050,-1510
C01807=1949,30608,-30383,956,-27054,-1512
C01808=1956,30616,-30374,955,-27057,-1515
C01809=1967,30610,-30381,954,-27055,-1519
C01810=1962,30600,-30393,954,-27051,-1518
C01811=1961,30587,-30409,955,-27047,-1517
C01812=1958,30575,-30424,955,-27042,-1516
C01813=1952,30563,-30437,956,-27038,-1514
C01814=1953,30550,-30453,956,-27033,-1515
C01815=1954,30537,-30469,956,-27028,-1515
C01816=1955,30524,-30485,956,-27023,-1516
C01817=1956,30511,-30501,956,-27019,-1516
C01818=1957,30498,-30517,956,-27014,-1517
C01819=1958,30485,-30532,956,-27009,-1517
C01820=1958,30473,-30547,956,-27004,-1517
C01821=1946,30467,-30553,958,-27002,-1512
C01822=1940,30456,-30567,959,-26998,-1510
C01823=1947,30446,-30579,958,-26994,-1513
C01824=1952,30435,-30592,958,-26990,-1515
C01825=1953,30422,-30608,958,-26986,-1515
C01826=1958,30411,-30621,957,-26982,-1518
C01827=1960,30402,-30632,957,-26978,-1519
C01828=1955,30390,-30646,958,-26974,-1517
C01829=1956,30377,-30662,958,-26969,-1517
C01830=1947,30366,-30675,959,-26965,-1514
C01831=1948,30353,-30691,959,-26960,-1514
C01832=1949,30340,-30707,959,-26955,-1515
C01833=1950,30327,-30723,959,-26951,-1515
C01834=1951,30314,-30738,959,-26946,-1516
C01835=1952,30301,-30754,959,-26941,-1516
C01836=1962,30293,-30764,958,-26938,-1520
C01837=1964,30280,-30779,958,-26933,-1521
C01838=1965,30267,-30795,958,-26929,-1521
C01839=1965,30267,-29395,958,-26929,-1521
C01840=1351,30193,-26887,1048,-26896,-1284
C01841=1351,30193,-30887,1048,-26896,-1284
C01842=1341,30192,-30889,1050,-26895,-1280
C01843=1331,30191,-30891,1051,-26895,-1276
C01844=1322,30189,-30893,1052,-26894,-1272
C01845=1312,30188,-30894,1054,-26894,-1269
C01846=1304,30193,-30888,1055,-26896,-1266
C01847=1296,30195,-30886,1056,-26896,-1262
C01848=1286,30194,-30887,1057,-26896,-1259
C01849=1277,30195,-30886,1059,-26896,-1255
C01850=1270,30201,-30879,1060,-26898,-1252
C01851=1263,30206,-30873,1061,-26900,-1250
C01852=1255,30211,-30866,1062,-26902,-1247
C01853=1248,30217,-30860,1063,-26904,-1244
C01854=1238,30215,-30862,1064,-26903,-1240
C01855=1231,30221,-30855,1065,-26905,-1237
C01856=1227,30228,-30847,1066,-26908,-1235
C01857=1223,30235,-30838,1066,-26910,-1234
C01858=1216,30241,-30831,1067,-26912,-1231
C01859=1215,30250,-30820,1067,-26915,-1231
C01860=1208,30255,-30814,1068,-26918,-1228
C01861=1204,30262,-30805,1069,-26920,-1226
C01862=1203,30271,-30794,1069,-26923,-1226
C01863=1203,30280,-30783,1068,-26927,-1226
C01864=1202,30289,-30772,1068,-26930,-1225
C01865=1202,30298,-30761,1068,-26933,-1225
C01866=1201,30308,-30751,1068,-26937,-1225
C01867=1200,30317,-30740,1068,-26940,-1224
C01868=1200,30326,-30729,1068,-26943,-1224
C01869=1200,30335,-30718,1068,-26947,-1224
C01870=1206,30342,-30709,1067,-26950,-1226
C01871=1208,30350,-30699,1067,-26953,-1227
C01872=1212,30351,-30698,1066,-26953,-1229
C01873=1219,30346,-30705,1065,-26951,-1231
C01874=1220,30336,-30715,1065,-26948,-1232
C01875=1220,30327,-30726,1065,-26944,-1232
C01876=1221,30318,-30737,1065,-26941,-1232
C01877=1215,30311,-30746,1066,-26938,-1230
C01878=1212,30303,-30756,1067,-26935,-1229
C01879=1212,30294,-30767,1067,-26932,-1229
C01880=1215,30286,-30776,1067,-26929,-1231
C01881=1223,30281,-30783,1066,-26927,-1233
C01882=1224,30272,-30793,1066,-26924,-1234
C01883=1225,30263,-30804,1066,-26920,-1234
C01884=1225,30254,-30815,1066,-26917,-1235
C01885=1231,30248,-30823,1065,-26915,-1237
C01886=1238,30242,-30829,1064,-26913,-1240
C01887=1246,30237,-30836,1063,-26911,-1243
C01888=1253,30231,-30842,1062,-26909,-1246
C01889=1258,30225,-30850,1061,-26907,-1248
C01890=1261,30217,-30860,1061,-26904,-1249
C01891=1268,30211,-30866,1060,-26902,-1251
C01892=1277,30211,-30866,1059,-26902,-1255
C01893=1285,30208,-30871,1057,-26901,-1258
C01894=1293,30204,-30875,1056,-26899,-1261
C01895=1303,30206,-30873,1055,-26900,-1265
C01896=1313,30207,-30871,1053,-26901,-1269
C01897=1322,30207,-30871,1052,-26901,-1273
C01898=1329,30202,-30877,1051,-26899,-1275
C01899=1338,30201,-30878,1050,-26899,-1279
C01900=1346,30198,-30882,1049,-26898,-1282
C01901=1351,30193,-30887,1048,-26896,-1284
C01902=1351,30193,-29487,1048,-26896,-1284
C01903=880,30355,-26695,1114,-26951,-1100
C01904=880,30355,-30695,1114,-26951,-1100
C01905=870,30353,-30697,1116,-26951,-1096
C01906=869,30363,-30685,1116,-26954,-1096
C01907=870,30373,-30674,1116,-26958,-1096
C01908=877,30381,-30664,1114,-26961,-1098
C01909=878,30391,-30652,1114,-26964,-1099
C01910=877,30401,-30640,1114,-26968,-1098
C01911=877,30411,-30628,1114,-26972,-1098
C01912=883,30419,-30618,1113,-26975,-1100
C01913=886,30428,-30607,1113,-26978,-1101
C01914=885,30438,-30595,1113,-26982,-1101
C01915=885,30448,-30583,1112,-26986,-1101
C01916=884,30458,-30571,1112,-26989,-1100
C01917=883,30468,-30559,1112,-26993,-1100
C01918=877,30475,-30551,1113,-26995,-1097
C01919=872,30483,-30541,1114,-26998,-1096
C01920=868,30490,-30532,1114,-27001,-1094
C01921=860,30496,-30525,1115,-27003,-1090
C01922=852,30502,-30517,1117,-27005,-1087
C01923=844,30508,-30510,1118,-27008,-1084
C01924=836,30514,-29103,1119,-27010,-1081
C01925=-41004,59868,4099,4900,-34257,16705
C01926=-41004,59868,1099,4900,-34257,16705
C01927=-41004,64596,1380,5213,-31659,16463
C01928=-41004,59868,1099,4900,-34257,16705
C01929=-41004,59868,9099,4900,-34257,16705
C01930=836,30514,-26503,1119,-27010,-1081
C01931=836,30514,-30503,1119,-27010,-1081
C01932=828,30520,-30496,1120,-27012,-1078
C01933=820,30526,-30489,1121,-27014,-1075
C01934=812,30532,-30482,1122,-27016,-1072
C01935=804,30538,-30474,1123,-27018,-1068
C01936=795,30543,-30469,1124,-27020,-1065
C01937=787,30544,-30468,1125,-27020,-1062
C01938=784,30553,-30457,1126,-27023,-1061
C01939=776,30559,-30450,1127,-27025,-1058
C01940=775,30568,-30438,1127,-27029,-1057
C01941=783,30562,-30445,1126,-27027,-1060
C01942=793,30562,-30446,1124,-27027,-1064
C01943=802,30558,-30451,1123,-27025,-1067
C01944=810,30552,-30458,1122,-27023,-1071
C01945=818,30546,-30465,1121,-27021,-1074
C01946=828,30547,-30464,1119,-27022,-1078
C01947=836,30541,-30471,1118,-27019,-1081
C01948=844,30535,-30478,1117,-27017,-1084
C01949=852,30529,-30485,1116,-27015,-1087
C01950=860,30523,-30492,1115,-27013,-1091
C01951=868,30517,-30500,1114,-27011,-1094
C01952=876,30511,-30507,1113,-27009,-1097
C01953=881,30503,-30516,1112,-27006,-1099
C01954=885,30495,-30526,1112,-27003,-1100
C01955=892,30489,-30533,1111,-27001,-1103
C01956=894,30480,-30545,1111,-26997,-1104
C01957=902,30474,-30552,1110,-26995,-1107
C01958=904,30464,-30563,1109,-26992,-1108
C01959=905,30454,-30575,1109,-26988,-1108
C01960=905,30444,-30587,1110,-26984,-1109
C01961=906,30434,-30599,1110,-26981,-1109
C01962=899,30426,-30609,1111,-26978,-1106
C01963=897,30417,-30620,1111,-26974,-1106
C01964=897,30407,-30633,1111,-26971,-1106
C01965=892,30398,-30643,1112,-26967,-1104
C01966=888,30389,-30654,1113,-26964,-1103
C01967=883,30384,-30661,1114,-26962,-1101
C01968=874,30378,-30667,1115,-26960,-1097
C01969=869,30370,-30677,1116,-26957,-1095
C01970=872,30361,-30688,1115,-26953,-1096
C01971=880,30355,-30695,1114,-26951,-1100
C01972=880,30355,-29295,1114,-26951,-1100
C01973=635,30348,-26705,1150,-26946,-1005
C01974=635,30348,-30705,1150,-26946,-1005
C01975=636,30335,-30721,1150,-26942,-1005
C01976=636,30322,-30736,1150,-26937,-1005
C01977=637,30310,-30751,1150,-26932,-1006
C01978=638,30297,-30767,1150,-26928,-1006
C01979=639,30284,-30782,1150,-26923,-1007
C01980=639,30271,-30797,1150,-26918,-1007
C01981=637,30259,-30812,1151,-26914,-1006
C01982=630,30249,-30825,1152,-26910,-1004
C01983=631,30236,-30840,1152,-26905,-1004
C01984=632,30223,-30856,1152,-26901,-1005
C01985=633,30210,-30871,1152,-26896,-1005
C01986=633,30198,-30886,1152,-26891,-1005
C01987=623,30193,-30892,1154,-26889,-1002
C01988=623,30206,-30877,1154,-26894,-1001
C01989=622,30218,-30861,1154,-26899,-1001
C01990=621,30231,-30846,1154,-26903,-1000
C01991=620,30244,-30831,1153,-26908,-1000
C01992=620,30257,-30815,1153,-26913,-1000
C01993=619,30269,-30800,1153,-26917,-999
C01994=618,30282,-30785,1153,-26922,-999
C01995=618,30295,-30769,1153,-26927,-998
C01996=617,30307,-30754,1153,-26931,-998
C01997=616,30320,-30739,1153,-26936,-998
C01998=615,30333,-30724,1153,-26941,-997
C01999=615,30345,-30708,1153,-26945,-997
C02000=614,30358,-30693,1153,-26950,-996
C02001=613,30371,-30678,1153,-26955,-996
C02002=612,30383,-30662,1153,-26959,-996
C02003=612,30396,-30647,1153,-26964,-995
C02004=611,30409,-30632,1153,-26969,-995
C02005=610,30421,-30616,1153,-26973,-994
C02006=606,30432,-30603,1153,-26977,-993
C02007=599,30441,-30592,1154,-26981,-990
C02008=593,30451,-30580,1155,-26984,-987
C02009=587,30461,-30568,1155,-26988,-985
C02010=580,30470,-30558,1156,-26991,-982
C02011=576,30481,-30544,1157,-26995,-981
C02012=567,30489,-30535,1158,-26998,-977
C02013=565,30501,-30520,1158,-27002,-976
C02014=560,30512,-30507,1159,-27006,-974
C02015=553,30521,-30496,1159,-27010,-971
C02016=553,30534,-30481,1159,-27014,-971
C02017=561,30530,-30486,1158,-27013,-974
C02018=564,30518,-30500,1158,-27009,-976
C02019=574,30511,-30509,1157,-27006,-980
C02020=577,30499,-30523,1156,-27002,-981
C02021=586,30491,-30533,1155,-26999,-984
C02022=591,30480,-30545,1155,-26995,-986
C02023=601,30473,-30554,1153,-26992,-990
C02024=608,30464,-30566,1152,-26989,-993
C02025=614,30454,-30577,1152,-26985,-995
C02026=619,30444,-30590,1151,-26982,-998
C02027=620,30431,-30605,1151,-26977,-998
C02028=630,30424,-30614,1150,-26974,-1002
C02029=631,30411,-30629,1150,-26970,-1003
C02030=632,30398,-30644,1150,-26965,-1003
C02031=633,30386,-30660,1150,-26960,-1003
C02032=633,30373,-30675,1150,-26956,-1004
C02033=634,30360,-30690,1150,-26951,-1004
C02034=635,30348,-30705,1150,-26946,-1005
C02035=635,30348,-29305,1150,-26946,-1005
C02036=402,30500,-26523,1182,-27000,-913
C02037=402,30500,-30523,1182,-27000,-913
C02038=371,31056,-29853,1178,-27204,-896
C02039=341,31611,-29183,1175,-27409,-878
C02040=310,32167,-28513,1172,-27613,-861
C02041=290,32713,-27855,1167,-27813,-848
C02042=260,33268,-27185,1164,-28017,-831
C02043=220,33819,-26521,1162,-28220,-811
C02044=189,34374,-25851,1159,-28424,-793
C02045=150,34925,-25187,1157,-28626,-773
C02046=119,35481,-24517,1153,-28830,-756
C02047=89,36036,-23847,1150,-29034,-739
C02048=483,36247,-23588,1094,-29118,-892
C02049=1028,36328,-23482,1019,-29157,-1107
C02050=1572,36409,-23377,944,-29195,-1321
C02051=2112,36499,-23261,870,-29237,-1533
C02052=2657,36580,-23156,795,-29276,-1748
C02053=3202,36661,-23050,720,-29314,-1962
C02054=3746,36742,-22945,645,-29353,-2176
C02055=4291,36823,-22840,571,-29391,-2391
C02056=4836,36904,-22735,496,-29430,-2605
C02057=5380,36985,-22629,421,-29468,-2819
C02058=5925,37066,-22524,346,-29507,-3033
C02059=6466,37131,-22438,272,-29540,-3246
C02060=6563,36597,-23087,260,-29340,-3285
C02061=6650,36047,-23754,249,-29134,-3320
C02062=6736,35497,-24422,238,-28928,-3355
C02063=6823,34947,-25089,228,-28723,-3390
C02064=6910,34397,-25757,217,-28517,-3425
C02065=6996,33848,-26424,206,-28311,-3460
C02066=7083,33298,-27092,196,-28106,-3494
C02067=7169,32748,-27759,185,-27900,-3529
C02068=7256,32198,-28426,174,-27694,-3564
C02069=7342,31648,-29094,164,-27489,-3599
C02070=7429,31099,-29761,153,-27283,-3634
C02071=7516,30549,-30429,142,-27077,-3669
C02072=7602,29999,-31096,132,-26872,-3703
C02073=7689,29449,-31764,121,-26666,-3738
C02074=7775,28899,-32431,110,-26460,-3773
C02075=7862,28349,-33099,100,-26255,-3808
C02076=7937,27802,-33763,91,-26050,-3838
C02077=8024,27252,-34431,80,-25844,-3873
C02078=7563,27059,-34665,151,-25770,-3697
C02079=6931,26969,-34774,248,-25734,-3456
C02080=6314,26871,-34893,342,-25695,-3219
C02081=5682,26781,-35002,439,-25659,-2977
C02082=5050,26691,-35112,535,-25622,-2736
C02083=4418,26601,-35221,632,-25586,-2494
C02084=3786,26510,-35331,728,-25550,-2252
C02085=3155,26420,-35440,825,-25514,-2010
C02086=2526,26340,-35537,921,-25481,-1769
C02087=1894,26250,-35647,1017,-25445,-1527
C02088=1263,26160,-35756,1114,-25409,-1286
C02089=645,26062,-35875,1208,-25370,-1049
C02090=615,26610,-35214,1205,-25571,-1032
C02091=584,27165,-34544,1202,-25775,-1015
C02092=554,27721,-33874,1198,-25979,-998
C02093=523,28277,-33204,1195,-26184,-981
C02094=493,28833,-32534,1192,-26388,-964
C02095=462,29388,-31863,1188,-26592,-947
C02096=432,29944,-31193,1185,-26796,-930
C02097=402,30500,-29123,1182,-27000,-913
C02098=-41004,59868,4099,4900,-34257,16705
C02099=-41004,59868,1099,4900,-34257,16705
C02100=-41004,64596,1380,5213,-31659,16463
C02101=-41004,59868,1099,4900,-34257,16705
C02102=-41004,59868,9099,4900,-34257,16705
C02103=402,30500,-26523,1182,-27000,-913
C02104=402,30500,-30523,1182,-27000,-913
C02105=402,30500,-29123,1182,-27000,-913
C02106=878,30754,-26214,1109,-27098,-1095
C02107=878,30754,-30214,1109,-27098,-1095
C02108=875,30764,-30202,1110,-27102,-1094
C02109=867,30771,-30193,1111,-27104,-1091
C02110=864,30781,-30181,1111,-27108,-1090
C02111=863,30792,-30168,1111,-27112,-1089
C02112=854,30798,-30160,1112,-27114,-1086
C02113=852,30809,-30148,1112,-27118,-1085
C02114=852,30820,-30134,1112,-27122,-1084
C02115=851,30831,-30121,1112,-27127,-1084
C02116=850,30842,-30107,1112,-27131,-1084
C02117=855,30843,-30107,1112,-27131,-1086
C02118=861,30834,-30117,1111,-27128,-1088
C02119=866,30826,-30127,1110,-27125,-1090
C02120=872,30817,-30137,1109,-27122,-1092
C02121=873,30806,-30151,1109,-27118,-1093
C02122=873,30795,-30164,1110,-27113,-1093
C02123=881,30788,-30173,1109,-27111,-1096
C02124=885,30778,-30184,1108,-27107,-1098
C02125=892,30770,-30194,1107,-27105,-1100
C02126=896,30761,-30205,1107,-27101,-1102
C02127=902,30753,-30214,1106,-27098,-1105
C02128=911,30747,-30222,1105,-27096,-1108
C02129=920,30740,-30230,1103,-27094,-1112
C02130=929,30733,-30238,1102,-27091,-1115
C02131=938,30727,-30246,1101,-27089,-1119
C02132=947,30720,-30254,1100,-27086,-1122
C02133=958,30719,-30255,1098,-27086,-1127
C02134=967,30714,-30262,1097,-27084,-1130
C02135=976,30707,-30270,1096,-27082,-1134
C02136=985,30700,-30278,1095,-27080,-1137
C02137=994,30694,-30286,1093,-27077,-1141
C02138=1003,30687,-30294,1092,-27075,-1144
C02139=1012,30680,-30301,1091,-27073,-1148
C02140=1021,30674,-30309,1090,-27070,-1152
C02141=1024,30664,-30321,1089,-27067,-1153
C02142=1025,30653,-30334,1089,-27063,-1153
C02143=1034,30646,-30343,1088,-27060,-1157
C02144=1036,30636,-30355,1088,-27056,-1158
C02145=1044,30629,-30363,1087,-27054,-1161
C02146=1048,30619,-30375,1087,-27050,-1162
C02147=1038,30616,-30379,1088,-27049,-1159
C02148=1029,30623,-30371,1089,-27051,-1155
C02149=1026,30633,-30359,1090,-27055,-1154
C02150=1018,30640,-30350,1091,-27058,-1151
C02151=1015,30650,-30338,1091,-27061,-1150
C02152=1007,30657,-30330,1092,-27064,-1146
C02153=1004,30667,-30318,1092,-27067,-1145
C02154=996,30674,-30309,1093,-27070,-1142
C02155=987,30681,-30301,1095,-27072,-1138
C02156=978,30688,-30293,1096,-27075,-1135
C02157=969,30694,-30285,1097,-27077,-1131
C02158=960,30700,-30278,1098,-27079,-1128
C02159=949,30700,-30278,1100,-27079,-1123
C02160=940,30707,-30270,1101,-27082,-1120
C02161=931,30714,-30262,1102,-27084,-1116
C02162=922,30720,-30254,1103,-27086,-1113
C02163=913,30727,-30246,1105,-27089,-1109
C02164=904,30734,-30238,1106,-27091,-1106
C02165=896,30740,-30230,1107,-27093,-1102
C02166=887,30747,-30222,1108,-27096,-1099
C02167=878,30754,-30214,1109,-27098,-1095
C02168=878,30754,-28814,1109,-27098,-1095
C02169=1512,30843,-26102,1017,-27137,-1341
C02170=1512,30843,-30102,1017,-27137,-1341
C02171=1512,30850,-30094,1017,-27140,-1341
C02172=1511,30857,-30085,1017,-27142,-1340
C02173=1511,30864,-30077,1017,-27145,-1340
C02174=1510,30871,-30069,1017,-27147,-1340
C02175=1511,30877,-30061,1016,-27150,-1340
C02176=1516,30883,-30054,1016,-27152,-1342
C02177=1521,30887,-30049,1015,-27153,-1344
C02178=1528,30888,-30048,1014,-27154,-1347
C02179=1534,30885,-30052,1013,-27153,-1349
C02180=1540,30880,-30057,1012,-27151,-1351
C02181=1540,30874,-30065,1012,-27149,-1352
C02182=1541,30867,-30073,1012,-27146,-1352
C02183=1542,30861,-30081,1012,-27144,-1353
C02184=1548,30857,-30086,1011,-27142,-1355
C02185=1553,30852,-30090,1011,-27141,-1357
C02186=1559,30848,-30095,1010,-27140,-1359
C02187=1565,30846,-30099,1009,-27139,-1361
C02188=1572,30847,-30097,1008,-27139,-1364
C02189=1579,30848,-30096,1007,-27139,-1367
C02190=1587,30849,-30095,1006,-27140,-1370
C02191=1594,30850,-30093,1005,-27140,-1373
C02192=1601,30851,-30092,1004,-27141,-1375
C02193=1608,30852,-30091,1003,-27141,-1378
C02194=1616,30853,-30090,1002,-27142,-1381
C02195=1623,30854,-30088,1001,-27142,-1384
C02196=1630,30855,-30087,999,-27143,-1387
C02197=1638,30856,-30086,998,-27143,-1390
C02198=1645,30857,-30084,997,-27144,-1392
C02199=1652,30858,-30083,996,-27144,-1395
C02200=1659,30859,-30082,995,-27145,-1398
C02201=1667,30860,-30080,994,-27145,-1401
C02202=1674,30861,-30079,993,-27145,-1404
C02203=1679,30857,-30084,992,-27144,-1406
C02204=1684,30853,-30089,992,-27143,-1408
C02205=1677,30852,-30090,993,-27142,-1405
C02206=1670,30851,-30091,994,-27142,-1402
C02207=1663,30850,-30093,995,-27141,-1399
C02208=1655,30849,-30094,996,-27141,-1397
C02209=1650,30844,-30100,997,-27139,-1395
C02210=1645,30839,-30107,997,-27137,-1393
C02211=1638,30837,-30108,998,-27136,-1390
C02212=1631,30836,-30110,1000,-27136,-1387
C02213=1624,30835,-30111,1001,-27135,-1384
C02214=1616,30834,-30112,1002,-27135,-1382
C02215=1609,30833,-30114,1003,-27134,-1379
C02216=1602,30832,-30115,1004,-27134,-1376
C02217=1595,30831,-30116,1005,-27133,-1373
C02218=1589,30835,-30112,1006,-27135,-1371
C02219=1583,30839,-30107,1006,-27136,-1369
C02220=1576,30838,-30108,1007,-27136,-1366
C02221=1569,30837,-30110,1009,-27135,-1363
C02222=1562,30836,-30111,1010,-27135,-1360
C02223=1554,30834,-30112,1011,-27134,-1357
C02224=1547,30833,-30114,1012,-27134,-1355
C02225=1540,30832,-30115,1013,-27133,-1352
C02226=1533,30832,-30115,1014,-27133,-1349
C02227=1527,30836,-30111,1015,-27135,-1347
C02228=1521,30839,-30107,1015,-27136,-1345
C02229=1514,30838,-30108,1016,-27135,-1342
C02230=1512,30843,-30102,1017,-27137,-1341
C02231=1512,30843,-28702,1017,-27137,-1341
C02232=1410,31129,-25758,1028,-27242,-1299
C02233=1410,31129,-29758,1028,-27242,-1299
C02234=1403,31128,-29759,1029,-27241,-1296
C02235=1396,31127,-29760,1030,-27241,-1293
C02236=1389,31126,-29762,1031,-27240,-1291
C02237=1381,31125,-29763,1032,-27240,-1288
C02238=1374,31124,-29764,1033,-27239,-1285
C02239=1367,31123,-29765,1034,-27239,-1282
C02240=1360,31122,-29767,1035,-27238,-1280
C02241=1360,31128,-29759,1035,-27241,-1279
C02242=1364,31132,-29755,1035,-27242,-1281
C02243=1371,31133,-29753,1033,-27243,-1284
C02244=1378,31134,-29752,1032,-27243,-1286
C02245=1383,31138,-29747,1032,-27245,-1288
C02246=1388,31143,-29740,1031,-27247,-1290
C02247=1394,31146,-29737,1030,-27248,-1293
C02248=1401,31147,-29736,1029,-27248,-1295
C02249=1408,31148,-29735,1028,-27249,-1298
C02250=1415,31149,-29734,1027,-27249,-1301
C02251=1423,31150,-29732,1026,-27249,-1304
C02252=1430,31151,-29731,1025,-27250,-1306
C02253=1437,31152,-29730,1024,-27250,-1309
C02254=1444,31153,-29728,1023,-27251,-1312
C02255=1451,31154,-29727,1022,-27251,-1315
C02256=1458,31155,-29726,1021,-27252,-1317
C02257=1465,31156,-29725,1020,-27252,-1320
C02258=1472,31157,-29723,1019,-27253,-1323
C02259=1479,31158,-29722,1018,-27253,-1326
C02260=1486,31159,-29721,1017,-27254,-1328
C02261=1493,31160,-29719,1016,-27254,-1331
C02262=1500,31161,-29718,1014,-27254,-1334
C02263=1507,31162,-29717,1013,-27255,-1336
C02264=1513,31160,-29720,1013,-27254,-1339
C02265=1519,31156,-29725,1012,-27253,-1341
C02266=1525,31155,-29725,1011,-27252,-1343
C02267=1532,31156,-29724,1010,-27253,-1346
C02268=1539,31157,-29723,1009,-27253,-1349
C02269=1546,31158,-29721,1008,-27254,-1352
C02270=1553,31157,-29723,1007,-27253,-1354
C02271=1558,31153,-29727,1006,-27252,-1356
C02272=1558,31150,-29731,1006,-27251,-1356
C02273=1551,31149,-28332,1007,-27251,-1354
C02274=-41004,59868,4099,4900,-34257,16705
C02275=-41004,59868,1099,4900,-34257,16705
C02276=-41004,64596,1380,5213,-31659,16463
C02277=-41004,59868,1099,4900,-34257,16705
C02278=-41004,59868,9099,4900,-34257,16705
C02279=1551,31149,-25732,1007,-27251,-1354
C02280=1551,31149,-29732,1007,-27251,-1354
C02281=1544,31148,-29733,1008,-27250,-1351
C02282=1537,31147,-29735,1009,-27250,-1348
C02283=1530,31146,-29736,1010,-27249,-1345
C02284=1523,31145,-29737,1011,-27249,-1343
C02285=1516,31144,-29738,1012,-27248,-1340
C02286=1509,31143,-29740,1013,-27248,-1337
C02287=1502,31142,-29741,1015,-27247,-1334
C02288=1495,31141,-29742,1016,-27247,-1332
C02289=1488,31140,-29744,1017,-27247,-1329
C02290=1481,31139,-29745,1018,-27246,-1326
C02291=1473,31138,-29746,1019,-27246,-1323
C02292=1466,31137,-29747,1020,-27245,-1321
C02293=1459,31136,-29749,1021,-27245,-1318
C02294=1452,31135,-29750,1022,-27244,-1315
C02295=1445,31134,-29751,1023,-27244,-1313
C02296=1438,31133,-29753,1024,-27243,-1310
C02297=1431,31132,-29754,1025,-27243,-1307
C02298=1424,31131,-29755,1026,-27243,-1304
C02299=1417,31130,-29756,1027,-27242,-1302
C02300=1410,31129,-29758,1028,-27242,-1299
C02301=1410,31129,-28358,1028,-27242,-1299
C02302=1396,32054,-24641,1019,-27583,-1286
C02303=1396,32054,-28641,1019,-27583,-1286
C02304=1382,32061,-28632,1021,-27585,-1280
C02305=1368,32066,-28626,1023,-27587,-1275
C02306=1368,32078,-28612,1022,-27592,-1274
C02307=1382,32073,-28618,1020,-27590,-1280
C02308=1395,32063,-28630,1019,-27586,-1285
C02309=1412,32065,-28627,1016,-27587,-1292
C02310=1429,32068,-28623,1014,-27589,-1299
C02311=1446,32070,-28620,1011,-27590,-1305
C02312=1464,32073,-28617,1009,-27591,-1312
C02313=1479,32079,-28609,1007,-27593,-1318
C02314=1493,32087,-28600,1004,-27596,-1323
C02315=1508,32094,-28592,1002,-27599,-1329
C02316=1523,32101,-28583,1000,-27602,-1335
C02317=1535,32112,-28569,998,-27606,-1339
C02318=1549,32121,-28558,996,-27609,-1345
C02319=1563,32128,-28550,994,-27612,-1350
C02320=1577,32137,-28539,992,-27616,-1356
C02321=1593,32142,-28532,990,-27618,-1362
C02322=1606,32151,-28522,987,-27621,-1367
C02323=1618,32163,-28508,986,-27626,-1372
C02324=1631,32174,-28494,984,-27630,-1376
C02325=1644,32183,-28483,982,-27633,-1381
C02326=1659,32190,-28474,979,-27636,-1387
C02327=1673,32199,-28463,977,-27640,-1392
C02328=1685,32211,-28449,976,-27644,-1397
C02329=1697,32222,-28436,974,-27648,-1402
C02330=1711,32231,-28424,972,-27652,-1407
C02331=1722,32244,-28408,970,-27657,-1411
C02332=1737,32251,-28400,968,-27660,-1417
C02333=1748,32265,-28383,966,-27665,-1421
C02334=1762,32272,-28375,964,-27667,-1427
C02335=1774,32277,-28369,962,-27669,-1431
C02336=1781,32263,-28385,961,-27664,-1434
C02337=1767,32256,-28394,963,-27662,-1429
C02338=1755,32243,-28410,965,-27657,-1424
C02339=1741,32236,-28418,967,-27654,-1419
C02340=1730,32222,-28435,969,-27649,-1414
C02341=1715,32215,-28444,971,-27646,-1409
C02342=1704,32202,-28459,973,-27641,-1404
C02343=1692,32189,-28476,975,-27636,-1400
C02344=1678,32181,-28485,977,-27633,-1395
C02345=1666,32169,-28499,979,-27629,-1390
C02346=1652,32161,-28509,981,-27625,-1385
C02347=1637,32154,-28518,983,-27623,-1379
C02348=1624,32144,-28530,985,-27619,-1374
C02349=1611,32134,-28543,987,-27615,-1369
C02350=1597,32127,-28551,989,-27612,-1363
C02351=1582,32119,-28561,991,-27609,-1358
C02352=1570,32108,-28574,993,-27605,-1353
C02353=1556,32099,-28585,995,-27601,-1348
C02354=1541,32092,-28593,997,-27599,-1342
C02355=1528,32082,-28605,999,-27595,-1337
C02356=1512,32078,-28611,1002,-27593,-1331
C02357=1499,32069,-28622,1004,-27589,-1326
C02358=1482,32066,-28625,1006,-27588,-1319
C02359=1464,32064,-28628,1009,-27587,-1312
C02360=1447,32061,-28632,1011,-27586,-1306
C02361=1430,32059,-28635,1014,-27585,-1299
C02362=1413,32056,-28638,1016,-27584,-1292
C02363=1396,32054,-28641,1019,-27583,-1286
C02364=1396,32054,-27241,1019,-27583,-1286
C02365=1268,32293,-24353,1034,-27670,-1234
C02366=1268,32293,-28353,1034,-27670,-1234
C02367=1230,32287,-28360,1039,-27667,-1219
C02368=1194,32292,-28355,1044,-27669,-1205
C02369=1156,32286,-28362,1050,-27666,-1190
C02370=1121,32290,-28357,1055,-27667,-1176
